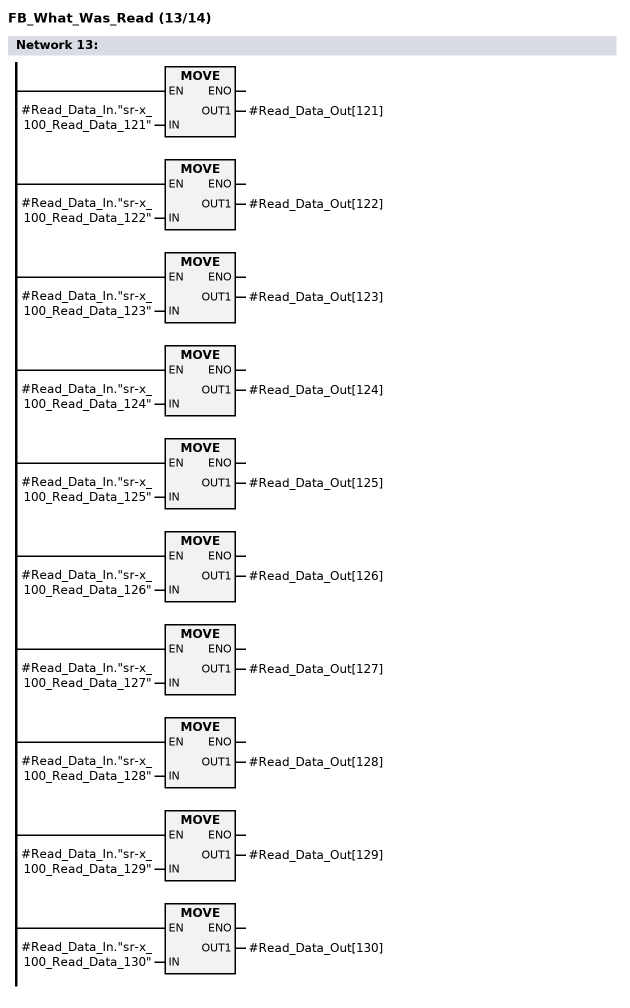
   RUNG wire#powerrail
      Move(in := #Read_Data_In."sr-x_100_Read_Data_121", out1 => #Read_Data_Out[121])
   END_RUNG
   RUNG wire#powerrail
      Move(in := #Read_Data_In."sr-x_100_Read_Data_122", out1 => #Read_Data_Out[122])
   END_RUNG
   RUNG wire#powerrail
      Move(in := #Read_Data_In."sr-x_100_Read_Data_123", out1 => #Read_Data_Out[123])
   END_RUNG
   RUNG wire#powerrail
      Move(in := #Read_Data_In."sr-x_100_Read_Data_124", out1 => #Read_Data_Out[124])
   END_RUNG
   RUNG wire#powerrail
      Move(in := #Read_Data_In."sr-x_100_Read_Data_125", out1 => #Read_Data_Out[125])
   END_RUNG
   RUNG wire#powerrail
      Move(in := #Read_Data_In."sr-x_100_Read_Data_126", out1 => #Read_Data_Out[126])
   END_RUNG
   RUNG wire#powerrail
      Move(in := #Read_Data_In."sr-x_100_Read_Data_127", out1 => #Read_Data_Out[127])
   END_RUNG
   RUNG wire#powerrail
      Move(in := #Read_Data_In."sr-x_100_Read_Data_128", out1 => #Read_Data_Out[128])
   END_RUNG
   RUNG wire#powerrail
      Move(in := #Read_Data_In."sr-x_100_Read_Data_129", out1 => #Read_Data_Out[129])
   END_RUNG
   RUNG wire#powerrail
      Move(in := #Read_Data_In."sr-x_100_Read_Data_130", out1 => #Read_Data_Out[130])
   END_RUNG
   // the same network as SCL:
   #Read_Data_Out[121] := #Read_Data_In."sr-x_100_Read_Data_121";
   #Read_Data_Out[122] := #Read_Data_In."sr-x_100_Read_Data_122";
   #Read_Data_Out[123] := #Read_Data_In."sr-x_100_Read_Data_123";
   #Read_Data_Out[124] := #Read_Data_In."sr-x_100_Read_Data_124";
   #Read_Data_Out[125] := #Read_Data_In."sr-x_100_Read_Data_125";
   #Read_Data_Out[126] := #Read_Data_In."sr-x_100_Read_Data_126";
   #Read_Data_Out[127] := #Read_Data_In."sr-x_100_Read_Data_127";
   #Read_Data_Out[128] := #Read_Data_In."sr-x_100_Read_Data_128";
   #Read_Data_Out[129] := #Read_Data_In."sr-x_100_Read_Data_129";
   #Read_Data_Out[130] := #Read_Data_In."sr-x_100_Read_Data_130";
END_REGION

REGION Network 14
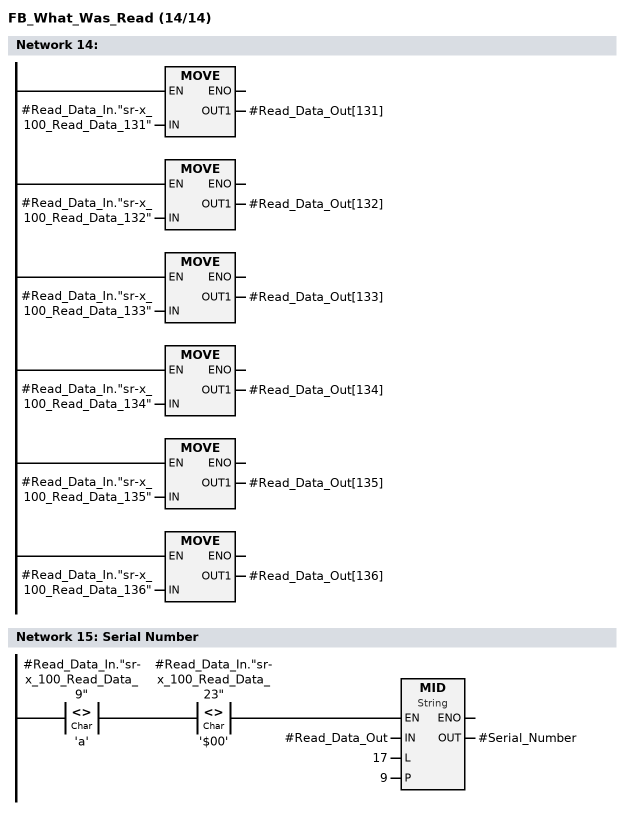
   RUNG wire#powerrail
      Move(in := #Read_Data_In."sr-x_100_Read_Data_131", out1 => #Read_Data_Out[131])
   END_RUNG
   RUNG wire#powerrail
      Move(in := #Read_Data_In."sr-x_100_Read_Data_132", out1 => #Read_Data_Out[132])
   END_RUNG
   RUNG wire#powerrail
      Move(in := #Read_Data_In."sr-x_100_Read_Data_133", out1 => #Read_Data_Out[133])
   END_RUNG
   RUNG wire#powerrail
      Move(in := #Read_Data_In."sr-x_100_Read_Data_134", out1 => #Read_Data_Out[134])
   END_RUNG
   RUNG wire#powerrail
      Move(in := #Read_Data_In."sr-x_100_Read_Data_135", out1 => #Read_Data_Out[135])
   END_RUNG
   RUNG wire#powerrail
      Move(in := #Read_Data_In."sr-x_100_Read_Data_136", out1 => #Read_Data_Out[136])
   END_RUNG
   // the same network as SCL:
   #Read_Data_Out[131] := #Read_Data_In."sr-x_100_Read_Data_131";
   #Read_Data_Out[132] := #Read_Data_In."sr-x_100_Read_Data_132";
   #Read_Data_Out[133] := #Read_Data_In."sr-x_100_Read_Data_133";
   #Read_Data_Out[134] := #Read_Data_In."sr-x_100_Read_Data_134";
   #Read_Data_Out[135] := #Read_Data_In."sr-x_100_Read_Data_135";
   #Read_Data_Out[136] := #Read_Data_In."sr-x_100_Read_Data_136";
END_REGION

REGION Network 15: Serial Number
   RUNG wire#powerrail
      { S7_Templates := "SrcType := Char" } NE_Contact(in1 := #Read_Data_In."sr-x_100_Read_Data_9", in2 := 'a')
      { S7_Templates := "SrcType := Char" } NE_Contact(in1 := #Read_Data_In."sr-x_100_Read_Data_23", in2 := '$00')
      { S7_Templates := "value_type := String" } MID(IN := #Read_Data_Out, L := 17, P := 9, OUT => #Serial_Number)
   END_RUNG
   // the same network as SCL:
   IF (#Read_Data_In."sr-x_100_Read_Data_9" <> 'a') AND (#Read_Data_In."sr-x_100_Read_Data_23" <> '$00') THEN
       MID(IN := #Read_Data_Out, L := 17, P := 9, OUT => #Serial_Number);
   END_IF;
END_REGION
END_FUNCTION_BLOCK

FUNCTION_BLOCK "FB_Marrige"   // FB8, LAD
{ S7_Optimized_Access := 'TRUE' }
// stored: MemoryReserve 100, SetENOAutomatically false
   VAR_INPUT
      In_Functional_Test_Odd : "IO_Device_Functinal_Test_Odd";
      In_Functional_Test_Even : "IO_Device_Functinal_Test_Even";
      Water_Fountain : String;
      Serial_Number : String[17];
      Read_Electrial_Voltage : UInt;
   END_VAR
   VAR_OUTPUT
      Functional_Tests_Panels : Array[0..31] of "Functional_Test";
      Got_Married : Bool;
   END_VAR
   VAR
      Aux_Trigger_0 : Bool;
      Aux_Trigger_1 : Bool;
      Aux_Trigger_2 : Bool;
      Aux_Trigger_3 : Bool;
      Aux_Trigger_4 : Bool;
      Aux_Trigger_5 : Bool;
      Aux_Trigger_6 : Bool;
      Aux_Trigger_7 : Bool;
      Aux_Trigger_8 : Bool;
      Aux_Trigger_9 : Bool;
      Aux_Trigger_10 : Bool;
      Aux_Trigger_11 : Bool;
      Aux_Trigger_12 : Bool;
      Aux_Trigger_13 : Bool;
      Aux_Trigger_14 : Bool;
      Aux_Trigger_15 : Bool;
      Aux_Trigger_16 : Bool;
      Aux_Trigger_17 : Bool;
      Aux_Trigger_18 : Bool;
      Aux_Trigger_19 : Bool;
      Aux_Trigger_20 : Bool;
      Aux_Trigger_21 : Bool;
      Aux_Trigger_22 : Bool;
      Aux_Trigger_23 : Bool;
      Aux_Trigger_24 : Bool;
      Aux_Trigger_25 : Bool;
      Aux_Trigger_26 : Bool;
      Aux_Trigger_27 : Bool;
      Aux_Trigger_28 : Bool;
      Aux_Trigger_29 : Bool;
      Aux_Trigger_30 : Bool;
      Aux_Trigger_31 : Bool;
   END_VAR
   VAR_TEMP   // added for the SCL form of the ladder/FBD networks
      _w1 : Bool;
   END_VAR
BEGIN

REGION Network 1: Panel 1
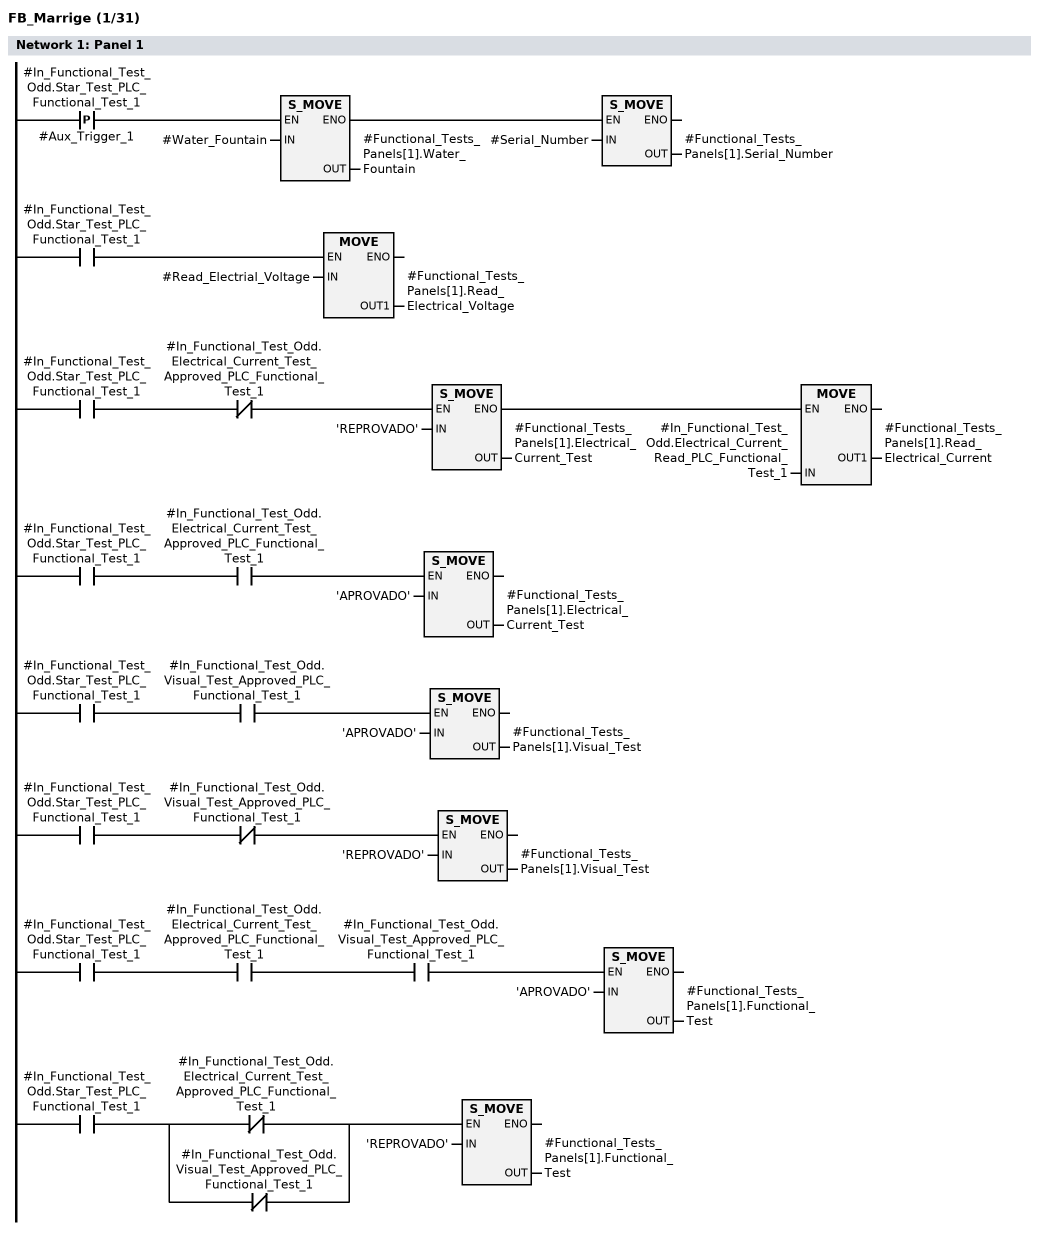
   RUNG wire#powerrail
      P_Contact(operand := #In_Functional_Test_Odd.Star_Test_PLC_Functional_Test_1, bit := #Aux_Trigger_1)
      S_Move(in := #Water_Fountain, out => #Functional_Tests_Panels[1].Water_Fountain)
      S_Move(in := #Serial_Number, out => #Functional_Tests_Panels[1].Serial_Number)
   END_RUNG
   RUNG wire#powerrail
      Contact( #In_Functional_Test_Odd.Star_Test_PLC_Functional_Test_1 )
      Move(in := #Read_Electrial_Voltage, out1 => #Functional_Tests_Panels[1].Read_Electrical_Voltage)
   END_RUNG
   RUNG wire#powerrail
      Contact( #In_Functional_Test_Odd.Star_Test_PLC_Functional_Test_1 )
      I_Contact( #In_Functional_Test_Odd.Electrical_Current_Test_Approved_PLC_Functional_Test_1 )
      S_Move(in := 'REPROVADO', out => #Functional_Tests_Panels[1].Electrical_Current_Test)
      Move(in := #In_Functional_Test_Odd.Electrical_Current_Read_PLC_Functional_Test_1, out1 => #Functional_Tests_Panels[1].Read_Electrical_Current)
   END_RUNG
   RUNG wire#powerrail
      Contact( #In_Functional_Test_Odd.Star_Test_PLC_Functional_Test_1 )
      Contact( #In_Functional_Test_Odd.Electrical_Current_Test_Approved_PLC_Functional_Test_1 )
      S_Move(in := 'APROVADO', out => #Functional_Tests_Panels[1].Electrical_Current_Test)
   END_RUNG
   RUNG wire#powerrail
      Contact( #In_Functional_Test_Odd.Star_Test_PLC_Functional_Test_1 )
      Contact( #In_Functional_Test_Odd.Visual_Test_Approved_PLC_Functional_Test_1 )
      S_Move(in := 'APROVADO', out => #Functional_Tests_Panels[1].Visual_Test)
   END_RUNG
   RUNG wire#powerrail
      Contact( #In_Functional_Test_Odd.Star_Test_PLC_Functional_Test_1 )
      I_Contact( #In_Functional_Test_Odd.Visual_Test_Approved_PLC_Functional_Test_1 )
      S_Move(in := 'REPROVADO', out => #Functional_Tests_Panels[1].Visual_Test)
   END_RUNG
   RUNG wire#powerrail
      Contact( #In_Functional_Test_Odd.Star_Test_PLC_Functional_Test_1 )
      Contact( #In_Functional_Test_Odd.Electrical_Current_Test_Approved_PLC_Functional_Test_1 )
      Contact( #In_Functional_Test_Odd.Visual_Test_Approved_PLC_Functional_Test_1 )
      S_Move(in := 'APROVADO', out => #Functional_Tests_Panels[1].Functional_Test)
   END_RUNG
   RUNG wire#powerrail
      Contact( #In_Functional_Test_Odd.Star_Test_PLC_Functional_Test_1 )
      wire#w1
      I_Contact( #In_Functional_Test_Odd.Electrical_Current_Test_Approved_PLC_Functional_Test_1 )
      wire#w2
      S_Move(in := 'REPROVADO', out => #Functional_Tests_Panels[1].Functional_Test)
   END_RUNG
   RUNG wire#w1
      I_Contact( #In_Functional_Test_Odd.Visual_Test_Approved_PLC_Functional_Test_1 )
   END_RUNG wire#w2
   // the same network as SCL:
   #_w1 := #In_Functional_Test_Odd.Star_Test_PLC_Functional_Test_1 AND NOT #Aux_Trigger_1;   // rising edge of #In_Functional_Test_Odd.Star_Test_PLC_Functional_Test_1
   #Aux_Trigger_1 := #In_Functional_Test_Odd.Star_Test_PLC_Functional_Test_1;
   IF #_w1 THEN
       #Functional_Tests_Panels[1].Water_Fountain := #Water_Fountain;
       #Functional_Tests_Panels[1].Serial_Number := #Serial_Number;
   END_IF;
   IF #In_Functional_Test_Odd.Star_Test_PLC_Functional_Test_1 THEN
       #Functional_Tests_Panels[1].Read_Electrical_Voltage := #Read_Electrial_Voltage;
   END_IF;
   IF #In_Functional_Test_Odd.Star_Test_PLC_Functional_Test_1 AND NOT #In_Functional_Test_Odd.Electrical_Current_Test_Approved_PLC_Functional_Test_1 THEN
       #Functional_Tests_Panels[1].Electrical_Current_Test := 'REPROVADO';
       #Functional_Tests_Panels[1].Read_Electrical_Current := #In_Functional_Test_Odd.Electrical_Current_Read_PLC_Functional_Test_1;
   END_IF;
   IF #In_Functional_Test_Odd.Star_Test_PLC_Functional_Test_1 AND #In_Functional_Test_Odd.Electrical_Current_Test_Approved_PLC_Functional_Test_1 THEN
       #Functional_Tests_Panels[1].Electrical_Current_Test := 'APROVADO';
   END_IF;
   IF #In_Functional_Test_Odd.Star_Test_PLC_Functional_Test_1 AND #In_Functional_Test_Odd.Visual_Test_Approved_PLC_Functional_Test_1 THEN
       #Functional_Tests_Panels[1].Visual_Test := 'APROVADO';
   END_IF;
   IF #In_Functional_Test_Odd.Star_Test_PLC_Functional_Test_1 AND NOT #In_Functional_Test_Odd.Visual_Test_Approved_PLC_Functional_Test_1 THEN
       #Functional_Tests_Panels[1].Visual_Test := 'REPROVADO';
   END_IF;
   IF #In_Functional_Test_Odd.Star_Test_PLC_Functional_Test_1 AND #In_Functional_Test_Odd.Electrical_Current_Test_Approved_PLC_Functional_Test_1 AND #In_Functional_Test_Odd.Visual_Test_Approved_PLC_Functional_Test_1 THEN
       #Functional_Tests_Panels[1].Functional_Test := 'APROVADO';
   END_IF;
   IF #In_Functional_Test_Odd.Star_Test_PLC_Functional_Test_1 AND (NOT #In_Functional_Test_Odd.Electrical_Current_Test_Approved_PLC_Functional_Test_1 OR NOT #In_Functional_Test_Odd.Visual_Test_Approved_PLC_Functional_Test_1) THEN
       #Functional_Tests_Panels[1].Functional_Test := 'REPROVADO';
   END_IF;
END_REGION

REGION Network 2: Panel 2
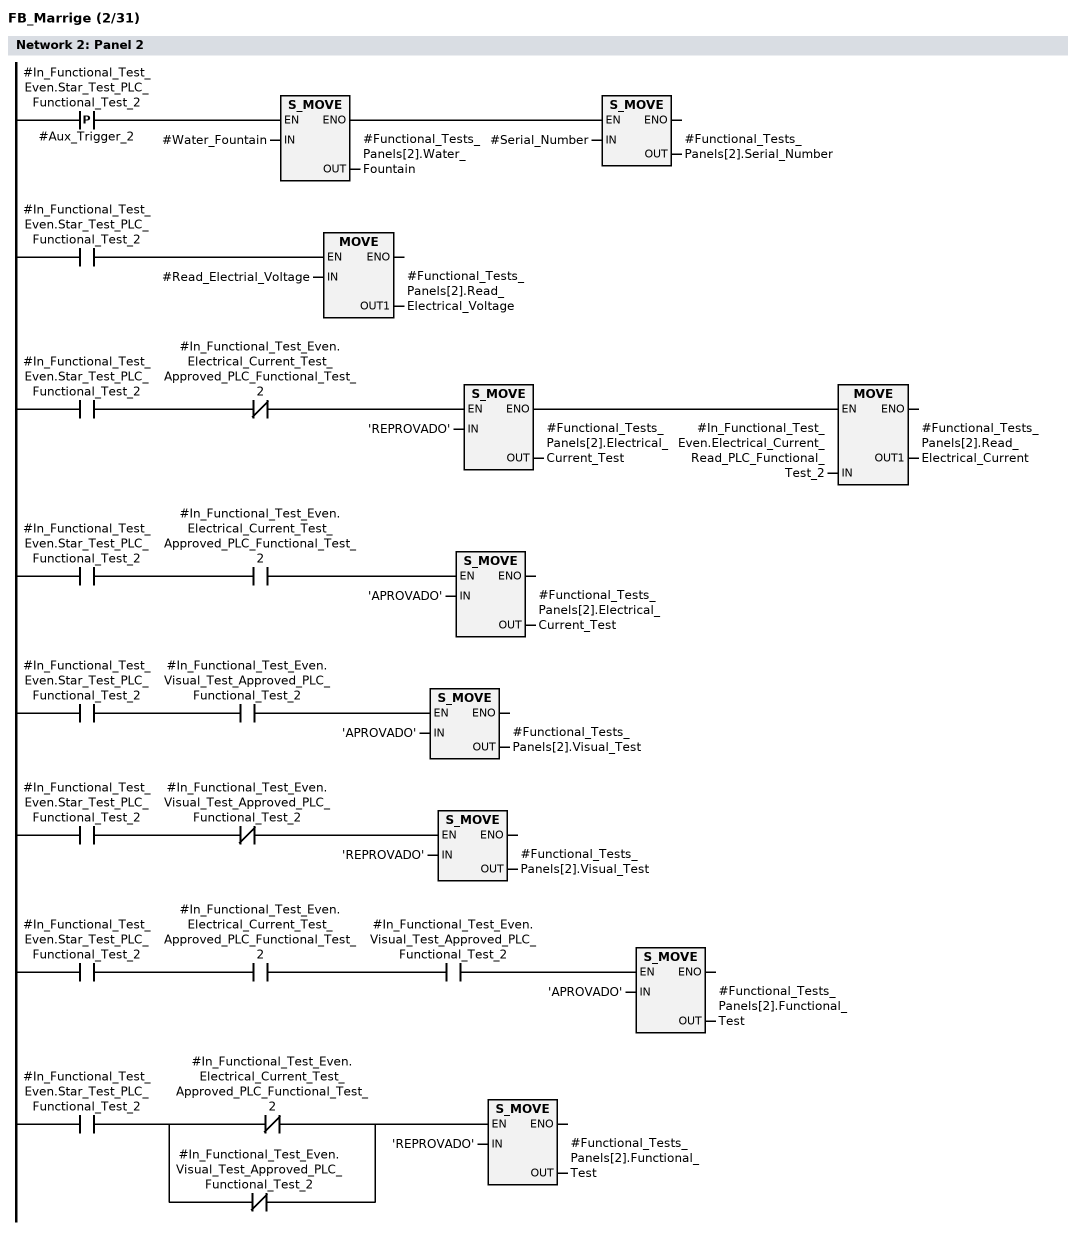
   RUNG wire#powerrail
      P_Contact(operand := #In_Functional_Test_Even.Star_Test_PLC_Functional_Test_2, bit := #Aux_Trigger_2)
      S_Move(in := #Water_Fountain, out => #Functional_Tests_Panels[2].Water_Fountain)
      S_Move(in := #Serial_Number, out => #Functional_Tests_Panels[2].Serial_Number)
   END_RUNG
   RUNG wire#powerrail
      Contact( #In_Functional_Test_Even.Star_Test_PLC_Functional_Test_2 )
      Move(in := #Read_Electrial_Voltage, out1 => #Functional_Tests_Panels[2].Read_Electrical_Voltage)
   END_RUNG
   RUNG wire#powerrail
      Contact( #In_Functional_Test_Even.Star_Test_PLC_Functional_Test_2 )
      I_Contact( #In_Functional_Test_Even.Electrical_Current_Test_Approved_PLC_Functional_Test_2 )
      S_Move(in := 'REPROVADO', out => #Functional_Tests_Panels[2].Electrical_Current_Test)
      Move(in := #In_Functional_Test_Even.Electrical_Current_Read_PLC_Functional_Test_2, out1 => #Functional_Tests_Panels[2].Read_Electrical_Current)
   END_RUNG
   RUNG wire#powerrail
      Contact( #In_Functional_Test_Even.Star_Test_PLC_Functional_Test_2 )
      Contact( #In_Functional_Test_Even.Electrical_Current_Test_Approved_PLC_Functional_Test_2 )
      S_Move(in := 'APROVADO', out => #Functional_Tests_Panels[2].Electrical_Current_Test)
   END_RUNG
   RUNG wire#powerrail
      Contact( #In_Functional_Test_Even.Star_Test_PLC_Functional_Test_2 )
      Contact( #In_Functional_Test_Even.Visual_Test_Approved_PLC_Functional_Test_2 )
      S_Move(in := 'APROVADO', out => #Functional_Tests_Panels[2].Visual_Test)
   END_RUNG
   RUNG wire#powerrail
      Contact( #In_Functional_Test_Even.Star_Test_PLC_Functional_Test_2 )
      I_Contact( #In_Functional_Test_Even.Visual_Test_Approved_PLC_Functional_Test_2 )
      S_Move(in := 'REPROVADO', out => #Functional_Tests_Panels[2].Visual_Test)
   END_RUNG
   RUNG wire#powerrail
      Contact( #In_Functional_Test_Even.Star_Test_PLC_Functional_Test_2 )
      Contact( #In_Functional_Test_Even.Electrical_Current_Test_Approved_PLC_Functional_Test_2 )
      Contact( #In_Functional_Test_Even.Visual_Test_Approved_PLC_Functional_Test_2 )
      S_Move(in := 'APROVADO', out => #Functional_Tests_Panels[2].Functional_Test)
   END_RUNG
   RUNG wire#powerrail
      Contact( #In_Functional_Test_Even.Star_Test_PLC_Functional_Test_2 )
      wire#w1
      I_Contact( #In_Functional_Test_Even.Electrical_Current_Test_Approved_PLC_Functional_Test_2 )
      wire#w2
      S_Move(in := 'REPROVADO', out => #Functional_Tests_Panels[2].Functional_Test)
   END_RUNG
   RUNG wire#w1
      I_Contact( #In_Functional_Test_Even.Visual_Test_Approved_PLC_Functional_Test_2 )
   END_RUNG wire#w2
   // the same network as SCL:
   #_w1 := #In_Functional_Test_Even.Star_Test_PLC_Functional_Test_2 AND NOT #Aux_Trigger_2;   // rising edge of #In_Functional_Test_Even.Star_Test_PLC_Functional_Test_2
   #Aux_Trigger_2 := #In_Functional_Test_Even.Star_Test_PLC_Functional_Test_2;
   IF #_w1 THEN
       #Functional_Tests_Panels[2].Water_Fountain := #Water_Fountain;
       #Functional_Tests_Panels[2].Serial_Number := #Serial_Number;
   END_IF;
   IF #In_Functional_Test_Even.Star_Test_PLC_Functional_Test_2 THEN
       #Functional_Tests_Panels[2].Read_Electrical_Voltage := #Read_Electrial_Voltage;
   END_IF;
   IF #In_Functional_Test_Even.Star_Test_PLC_Functional_Test_2 AND NOT #In_Functional_Test_Even.Electrical_Current_Test_Approved_PLC_Functional_Test_2 THEN
       #Functional_Tests_Panels[2].Electrical_Current_Test := 'REPROVADO';
       #Functional_Tests_Panels[2].Read_Electrical_Current := #In_Functional_Test_Even.Electrical_Current_Read_PLC_Functional_Test_2;
   END_IF;
   IF #In_Functional_Test_Even.Star_Test_PLC_Functional_Test_2 AND #In_Functional_Test_Even.Electrical_Current_Test_Approved_PLC_Functional_Test_2 THEN
       #Functional_Tests_Panels[2].Electrical_Current_Test := 'APROVADO';
   END_IF;
   IF #In_Functional_Test_Even.Star_Test_PLC_Functional_Test_2 AND #In_Functional_Test_Even.Visual_Test_Approved_PLC_Functional_Test_2 THEN
       #Functional_Tests_Panels[2].Visual_Test := 'APROVADO';
   END_IF;
   IF #In_Functional_Test_Even.Star_Test_PLC_Functional_Test_2 AND NOT #In_Functional_Test_Even.Visual_Test_Approved_PLC_Functional_Test_2 THEN
       #Functional_Tests_Panels[2].Visual_Test := 'REPROVADO';
   END_IF;
   IF #In_Functional_Test_Even.Star_Test_PLC_Functional_Test_2 AND #In_Functional_Test_Even.Electrical_Current_Test_Approved_PLC_Functional_Test_2 AND #In_Functional_Test_Even.Visual_Test_Approved_PLC_Functional_Test_2 THEN
       #Functional_Tests_Panels[2].Functional_Test := 'APROVADO';
   END_IF;
   IF #In_Functional_Test_Even.Star_Test_PLC_Functional_Test_2 AND (NOT #In_Functional_Test_Even.Electrical_Current_Test_Approved_PLC_Functional_Test_2 OR NOT #In_Functional_Test_Even.Visual_Test_Approved_PLC_Functional_Test_2) THEN
       #Functional_Tests_Panels[2].Functional_Test := 'REPROVADO';
   END_IF;
END_REGION

REGION Network 3: Panel 3
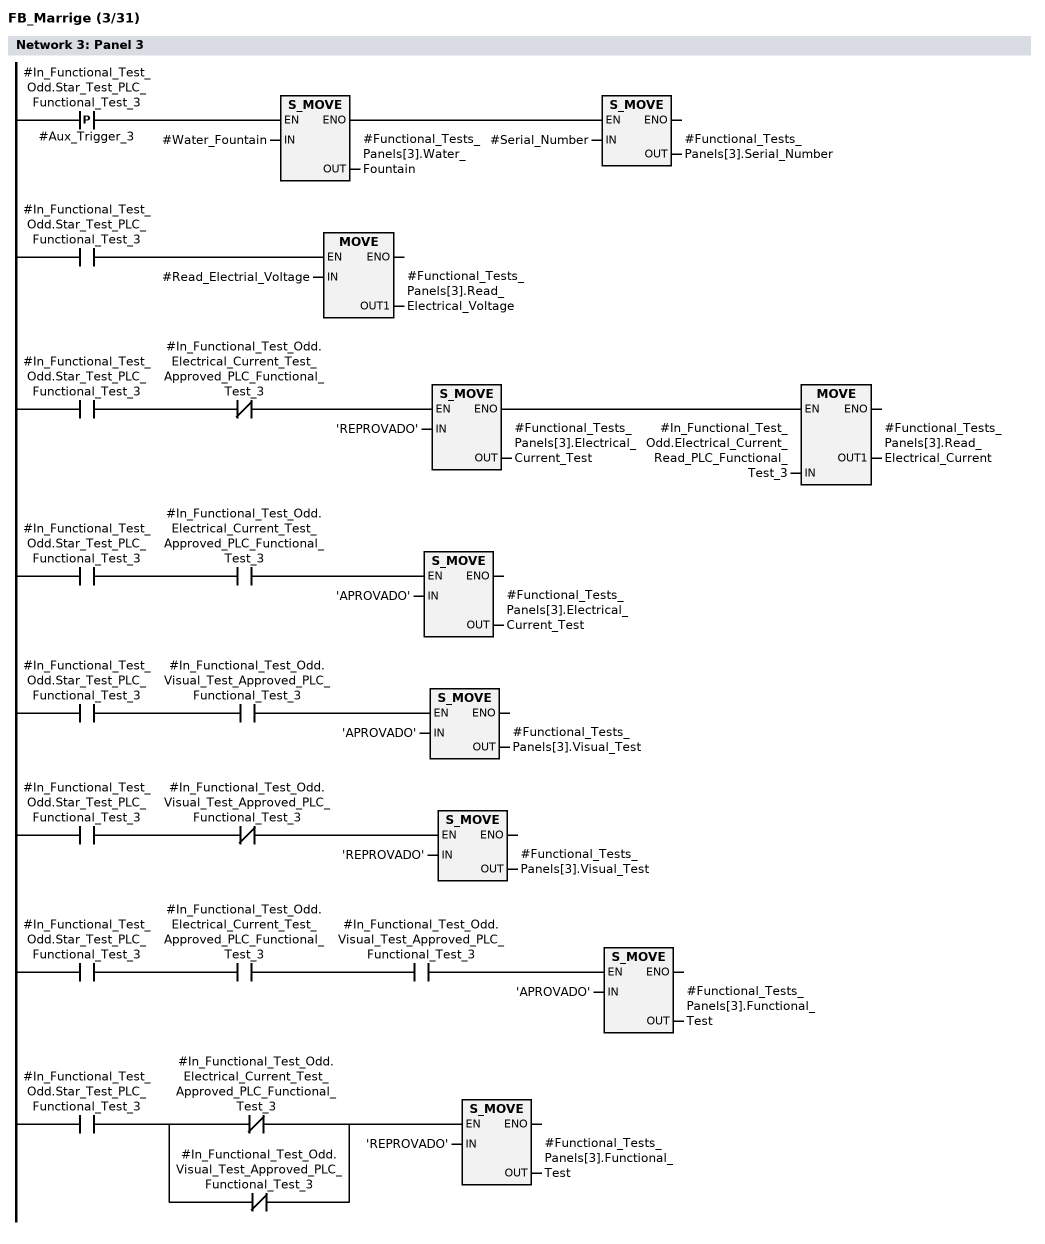
   RUNG wire#powerrail
      P_Contact(operand := #In_Functional_Test_Odd.Star_Test_PLC_Functional_Test_3, bit := #Aux_Trigger_3)
      S_Move(in := #Water_Fountain, out => #Functional_Tests_Panels[3].Water_Fountain)
      S_Move(in := #Serial_Number, out => #Functional_Tests_Panels[3].Serial_Number)
   END_RUNG
   RUNG wire#powerrail
      Contact( #In_Functional_Test_Odd.Star_Test_PLC_Functional_Test_3 )
      Move(in := #Read_Electrial_Voltage, out1 => #Functional_Tests_Panels[3].Read_Electrical_Voltage)
   END_RUNG
   RUNG wire#powerrail
      Contact( #In_Functional_Test_Odd.Star_Test_PLC_Functional_Test_3 )
      I_Contact( #In_Functional_Test_Odd.Electrical_Current_Test_Approved_PLC_Functional_Test_3 )
      S_Move(in := 'REPROVADO', out => #Functional_Tests_Panels[3].Electrical_Current_Test)
      Move(in := #In_Functional_Test_Odd.Electrical_Current_Read_PLC_Functional_Test_3, out1 => #Functional_Tests_Panels[3].Read_Electrical_Current)
   END_RUNG
   RUNG wire#powerrail
      Contact( #In_Functional_Test_Odd.Star_Test_PLC_Functional_Test_3 )
      Contact( #In_Functional_Test_Odd.Electrical_Current_Test_Approved_PLC_Functional_Test_3 )
      S_Move(in := 'APROVADO', out => #Functional_Tests_Panels[3].Electrical_Current_Test)
   END_RUNG
   RUNG wire#powerrail
      Contact( #In_Functional_Test_Odd.Star_Test_PLC_Functional_Test_3 )
      Contact( #In_Functional_Test_Odd.Visual_Test_Approved_PLC_Functional_Test_3 )
      S_Move(in := 'APROVADO', out => #Functional_Tests_Panels[3].Visual_Test)
   END_RUNG
   RUNG wire#powerrail
      Contact( #In_Functional_Test_Odd.Star_Test_PLC_Functional_Test_3 )
      I_Contact( #In_Functional_Test_Odd.Visual_Test_Approved_PLC_Functional_Test_3 )
      S_Move(in := 'REPROVADO', out => #Functional_Tests_Panels[3].Visual_Test)
   END_RUNG
   RUNG wire#powerrail
      Contact( #In_Functional_Test_Odd.Star_Test_PLC_Functional_Test_3 )
      Contact( #In_Functional_Test_Odd.Electrical_Current_Test_Approved_PLC_Functional_Test_3 )
      Contact( #In_Functional_Test_Odd.Visual_Test_Approved_PLC_Functional_Test_3 )
      S_Move(in := 'APROVADO', out => #Functional_Tests_Panels[3].Functional_Test)
   END_RUNG
   RUNG wire#powerrail
      Contact( #In_Functional_Test_Odd.Star_Test_PLC_Functional_Test_3 )
      wire#w1
      I_Contact( #In_Functional_Test_Odd.Electrical_Current_Test_Approved_PLC_Functional_Test_3 )
      wire#w2
      S_Move(in := 'REPROVADO', out => #Functional_Tests_Panels[3].Functional_Test)
   END_RUNG
   RUNG wire#w1
      I_Contact( #In_Functional_Test_Odd.Visual_Test_Approved_PLC_Functional_Test_3 )
   END_RUNG wire#w2
   // the same network as SCL:
   #_w1 := #In_Functional_Test_Odd.Star_Test_PLC_Functional_Test_3 AND NOT #Aux_Trigger_3;   // rising edge of #In_Functional_Test_Odd.Star_Test_PLC_Functional_Test_3
   #Aux_Trigger_3 := #In_Functional_Test_Odd.Star_Test_PLC_Functional_Test_3;
   IF #_w1 THEN
       #Functional_Tests_Panels[3].Water_Fountain := #Water_Fountain;
       #Functional_Tests_Panels[3].Serial_Number := #Serial_Number;
   END_IF;
   IF #In_Functional_Test_Odd.Star_Test_PLC_Functional_Test_3 THEN
       #Functional_Tests_Panels[3].Read_Electrical_Voltage := #Read_Electrial_Voltage;
   END_IF;
   IF #In_Functional_Test_Odd.Star_Test_PLC_Functional_Test_3 AND NOT #In_Functional_Test_Odd.Electrical_Current_Test_Approved_PLC_Functional_Test_3 THEN
       #Functional_Tests_Panels[3].Electrical_Current_Test := 'REPROVADO';
       #Functional_Tests_Panels[3].Read_Electrical_Current := #In_Functional_Test_Odd.Electrical_Current_Read_PLC_Functional_Test_3;
   END_IF;
   IF #In_Functional_Test_Odd.Star_Test_PLC_Functional_Test_3 AND #In_Functional_Test_Odd.Electrical_Current_Test_Approved_PLC_Functional_Test_3 THEN
       #Functional_Tests_Panels[3].Electrical_Current_Test := 'APROVADO';
   END_IF;
   IF #In_Functional_Test_Odd.Star_Test_PLC_Functional_Test_3 AND #In_Functional_Test_Odd.Visual_Test_Approved_PLC_Functional_Test_3 THEN
       #Functional_Tests_Panels[3].Visual_Test := 'APROVADO';
   END_IF;
   IF #In_Functional_Test_Odd.Star_Test_PLC_Functional_Test_3 AND NOT #In_Functional_Test_Odd.Visual_Test_Approved_PLC_Functional_Test_3 THEN
       #Functional_Tests_Panels[3].Visual_Test := 'REPROVADO';
   END_IF;
   IF #In_Functional_Test_Odd.Star_Test_PLC_Functional_Test_3 AND #In_Functional_Test_Odd.Electrical_Current_Test_Approved_PLC_Functional_Test_3 AND #In_Functional_Test_Odd.Visual_Test_Approved_PLC_Functional_Test_3 THEN
       #Functional_Tests_Panels[3].Functional_Test := 'APROVADO';
   END_IF;
   IF #In_Functional_Test_Odd.Star_Test_PLC_Functional_Test_3 AND (NOT #In_Functional_Test_Odd.Electrical_Current_Test_Approved_PLC_Functional_Test_3 OR NOT #In_Functional_Test_Odd.Visual_Test_Approved_PLC_Functional_Test_3) THEN
       #Functional_Tests_Panels[3].Functional_Test := 'REPROVADO';
   END_IF;
END_REGION

REGION Network 4: Panel 4
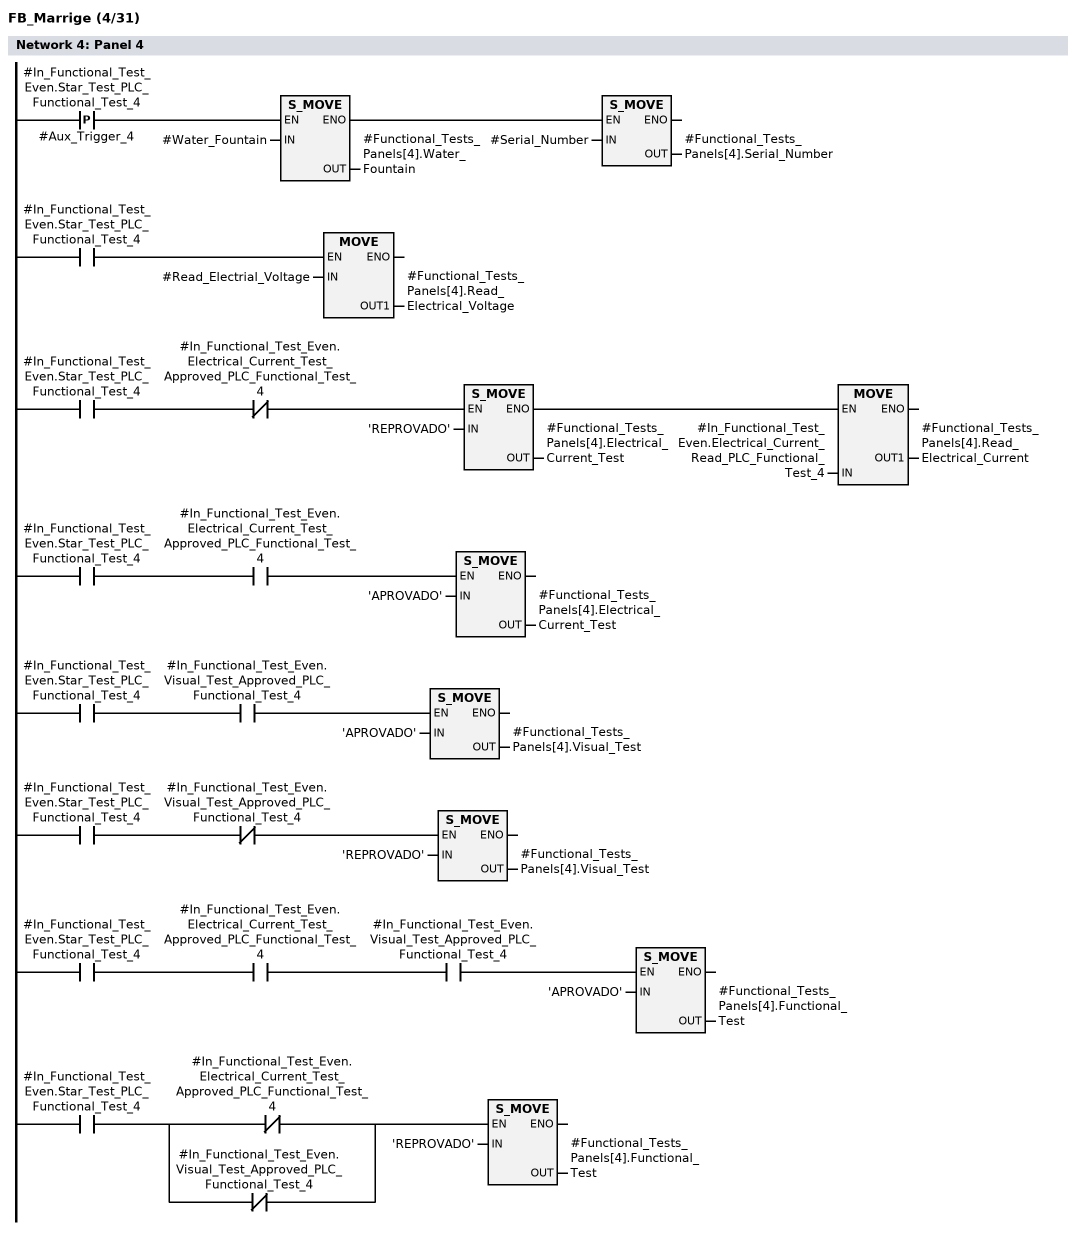
   RUNG wire#powerrail
      P_Contact(operand := #In_Functional_Test_Even.Star_Test_PLC_Functional_Test_4, bit := #Aux_Trigger_4)
      S_Move(in := #Water_Fountain, out => #Functional_Tests_Panels[4].Water_Fountain)
      S_Move(in := #Serial_Number, out => #Functional_Tests_Panels[4].Serial_Number)
   END_RUNG
   RUNG wire#powerrail
      Contact( #In_Functional_Test_Even.Star_Test_PLC_Functional_Test_4 )
      Move(in := #Read_Electrial_Voltage, out1 => #Functional_Tests_Panels[4].Read_Electrical_Voltage)
   END_RUNG
   RUNG wire#powerrail
      Contact( #In_Functional_Test_Even.Star_Test_PLC_Functional_Test_4 )
      I_Contact( #In_Functional_Test_Even.Electrical_Current_Test_Approved_PLC_Functional_Test_4 )
      S_Move(in := 'REPROVADO', out => #Functional_Tests_Panels[4].Electrical_Current_Test)
      Move(in := #In_Functional_Test_Even.Electrical_Current_Read_PLC_Functional_Test_4, out1 => #Functional_Tests_Panels[4].Read_Electrical_Current)
   END_RUNG
   RUNG wire#powerrail
      Contact( #In_Functional_Test_Even.Star_Test_PLC_Functional_Test_4 )
      Contact( #In_Functional_Test_Even.Electrical_Current_Test_Approved_PLC_Functional_Test_4 )
      S_Move(in := 'APROVADO', out => #Functional_Tests_Panels[4].Electrical_Current_Test)
   END_RUNG
   RUNG wire#powerrail
      Contact( #In_Functional_Test_Even.Star_Test_PLC_Functional_Test_4 )
      Contact( #In_Functional_Test_Even.Visual_Test_Approved_PLC_Functional_Test_4 )
      S_Move(in := 'APROVADO', out => #Functional_Tests_Panels[4].Visual_Test)
   END_RUNG
   RUNG wire#powerrail
      Contact( #In_Functional_Test_Even.Star_Test_PLC_Functional_Test_4 )
      I_Contact( #In_Functional_Test_Even.Visual_Test_Approved_PLC_Functional_Test_4 )
      S_Move(in := 'REPROVADO', out => #Functional_Tests_Panels[4].Visual_Test)
   END_RUNG
   RUNG wire#powerrail
      Contact( #In_Functional_Test_Even.Star_Test_PLC_Functional_Test_4 )
      Contact( #In_Functional_Test_Even.Electrical_Current_Test_Approved_PLC_Functional_Test_4 )
      Contact( #In_Functional_Test_Even.Visual_Test_Approved_PLC_Functional_Test_4 )
      S_Move(in := 'APROVADO', out => #Functional_Tests_Panels[4].Functional_Test)
   END_RUNG
   RUNG wire#powerrail
      Contact( #In_Functional_Test_Even.Star_Test_PLC_Functional_Test_4 )
      wire#w1
      I_Contact( #In_Functional_Test_Even.Electrical_Current_Test_Approved_PLC_Functional_Test_4 )
      wire#w2
      S_Move(in := 'REPROVADO', out => #Functional_Tests_Panels[4].Functional_Test)
   END_RUNG
   RUNG wire#w1
      I_Contact( #In_Functional_Test_Even.Visual_Test_Approved_PLC_Functional_Test_4 )
   END_RUNG wire#w2
   // the same network as SCL:
   #_w1 := #In_Functional_Test_Even.Star_Test_PLC_Functional_Test_4 AND NOT #Aux_Trigger_4;   // rising edge of #In_Functional_Test_Even.Star_Test_PLC_Functional_Test_4
   #Aux_Trigger_4 := #In_Functional_Test_Even.Star_Test_PLC_Functional_Test_4;
   IF #_w1 THEN
       #Functional_Tests_Panels[4].Water_Fountain := #Water_Fountain;
       #Functional_Tests_Panels[4].Serial_Number := #Serial_Number;
   END_IF;
   IF #In_Functional_Test_Even.Star_Test_PLC_Functional_Test_4 THEN
       #Functional_Tests_Panels[4].Read_Electrical_Voltage := #Read_Electrial_Voltage;
   END_IF;
   IF #In_Functional_Test_Even.Star_Test_PLC_Functional_Test_4 AND NOT #In_Functional_Test_Even.Electrical_Current_Test_Approved_PLC_Functional_Test_4 THEN
       #Functional_Tests_Panels[4].Electrical_Current_Test := 'REPROVADO';
       #Functional_Tests_Panels[4].Read_Electrical_Current := #In_Functional_Test_Even.Electrical_Current_Read_PLC_Functional_Test_4;
   END_IF;
   IF #In_Functional_Test_Even.Star_Test_PLC_Functional_Test_4 AND #In_Functional_Test_Even.Electrical_Current_Test_Approved_PLC_Functional_Test_4 THEN
       #Functional_Tests_Panels[4].Electrical_Current_Test := 'APROVADO';
   END_IF;
   IF #In_Functional_Test_Even.Star_Test_PLC_Functional_Test_4 AND #In_Functional_Test_Even.Visual_Test_Approved_PLC_Functional_Test_4 THEN
       #Functional_Tests_Panels[4].Visual_Test := 'APROVADO';
   END_IF;
   IF #In_Functional_Test_Even.Star_Test_PLC_Functional_Test_4 AND NOT #In_Functional_Test_Even.Visual_Test_Approved_PLC_Functional_Test_4 THEN
       #Functional_Tests_Panels[4].Visual_Test := 'REPROVADO';
   END_IF;
   IF #In_Functional_Test_Even.Star_Test_PLC_Functional_Test_4 AND #In_Functional_Test_Even.Electrical_Current_Test_Approved_PLC_Functional_Test_4 AND #In_Functional_Test_Even.Visual_Test_Approved_PLC_Functional_Test_4 THEN
       #Functional_Tests_Panels[4].Functional_Test := 'APROVADO';
   END_IF;
   IF #In_Functional_Test_Even.Star_Test_PLC_Functional_Test_4 AND (NOT #In_Functional_Test_Even.Electrical_Current_Test_Approved_PLC_Functional_Test_4 OR NOT #In_Functional_Test_Even.Visual_Test_Approved_PLC_Functional_Test_4) THEN
       #Functional_Tests_Panels[4].Functional_Test := 'REPROVADO';
   END_IF;
END_REGION

REGION Network 5: Panel 5
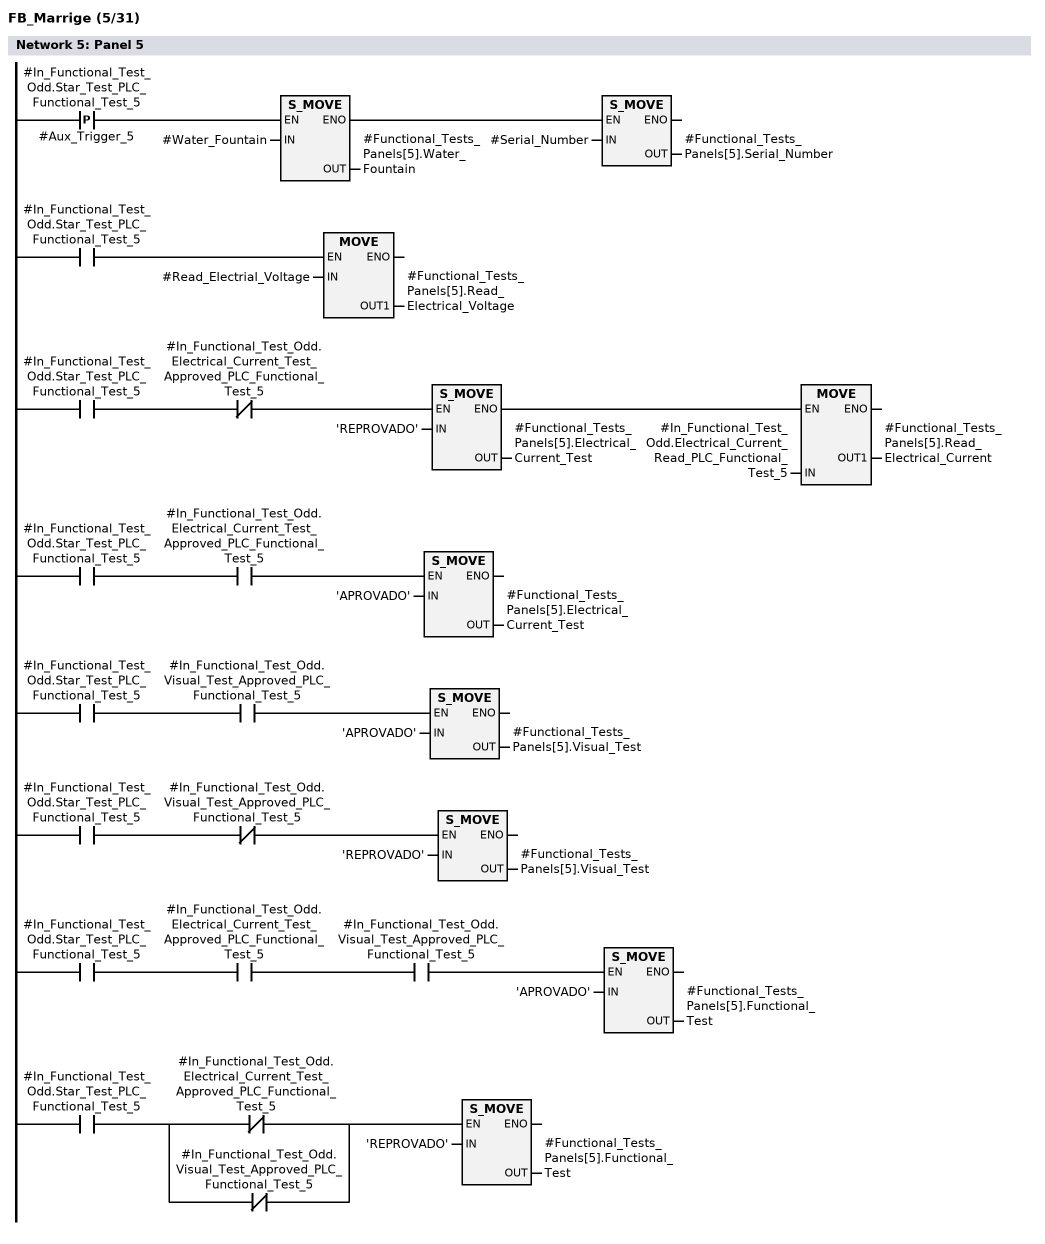
   RUNG wire#powerrail
      P_Contact(operand := #In_Functional_Test_Odd.Star_Test_PLC_Functional_Test_5, bit := #Aux_Trigger_5)
      S_Move(in := #Water_Fountain, out => #Functional_Tests_Panels[5].Water_Fountain)
      S_Move(in := #Serial_Number, out => #Functional_Tests_Panels[5].Serial_Number)
   END_RUNG
   RUNG wire#powerrail
      Contact( #In_Functional_Test_Odd.Star_Test_PLC_Functional_Test_5 )
      Move(in := #Read_Electrial_Voltage, out1 => #Functional_Tests_Panels[5].Read_Electrical_Voltage)
   END_RUNG
   RUNG wire#powerrail
      Contact( #In_Functional_Test_Odd.Star_Test_PLC_Functional_Test_5 )
      I_Contact( #In_Functional_Test_Odd.Electrical_Current_Test_Approved_PLC_Functional_Test_5 )
      S_Move(in := 'REPROVADO', out => #Functional_Tests_Panels[5].Electrical_Current_Test)
      Move(in := #In_Functional_Test_Odd.Electrical_Current_Read_PLC_Functional_Test_5, out1 => #Functional_Tests_Panels[5].Read_Electrical_Current)
   END_RUNG
   RUNG wire#powerrail
      Contact( #In_Functional_Test_Odd.Star_Test_PLC_Functional_Test_5 )
      Contact( #In_Functional_Test_Odd.Electrical_Current_Test_Approved_PLC_Functional_Test_5 )
      S_Move(in := 'APROVADO', out => #Functional_Tests_Panels[5].Electrical_Current_Test)
   END_RUNG
   RUNG wire#powerrail
      Contact( #In_Functional_Test_Odd.Star_Test_PLC_Functional_Test_5 )
      Contact( #In_Functional_Test_Odd.Visual_Test_Approved_PLC_Functional_Test_5 )
      S_Move(in := 'APROVADO', out => #Functional_Tests_Panels[5].Visual_Test)
   END_RUNG
   RUNG wire#powerrail
      Contact( #In_Functional_Test_Odd.Star_Test_PLC_Functional_Test_5 )
      I_Contact( #In_Functional_Test_Odd.Visual_Test_Approved_PLC_Functional_Test_5 )
      S_Move(in := 'REPROVADO', out => #Functional_Tests_Panels[5].Visual_Test)
   END_RUNG
   RUNG wire#powerrail
      Contact( #In_Functional_Test_Odd.Star_Test_PLC_Functional_Test_5 )
      Contact( #In_Functional_Test_Odd.Electrical_Current_Test_Approved_PLC_Functional_Test_5 )
      Contact( #In_Functional_Test_Odd.Visual_Test_Approved_PLC_Functional_Test_5 )
      S_Move(in := 'APROVADO', out => #Functional_Tests_Panels[5].Functional_Test)
   END_RUNG
   RUNG wire#powerrail
      Contact( #In_Functional_Test_Odd.Star_Test_PLC_Functional_Test_5 )
      wire#w1
      I_Contact( #In_Functional_Test_Odd.Electrical_Current_Test_Approved_PLC_Functional_Test_5 )
      wire#w2
      S_Move(in := 'REPROVADO', out => #Functional_Tests_Panels[5].Functional_Test)
   END_RUNG
   RUNG wire#w1
      I_Contact( #In_Functional_Test_Odd.Visual_Test_Approved_PLC_Functional_Test_5 )
   END_RUNG wire#w2
   // the same network as SCL:
   #_w1 := #In_Functional_Test_Odd.Star_Test_PLC_Functional_Test_5 AND NOT #Aux_Trigger_5;   // rising edge of #In_Functional_Test_Odd.Star_Test_PLC_Functional_Test_5
   #Aux_Trigger_5 := #In_Functional_Test_Odd.Star_Test_PLC_Functional_Test_5;
   IF #_w1 THEN
       #Functional_Tests_Panels[5].Water_Fountain := #Water_Fountain;
       #Functional_Tests_Panels[5].Serial_Number := #Serial_Number;
   END_IF;
   IF #In_Functional_Test_Odd.Star_Test_PLC_Functional_Test_5 THEN
       #Functional_Tests_Panels[5].Read_Electrical_Voltage := #Read_Electrial_Voltage;
   END_IF;
   IF #In_Functional_Test_Odd.Star_Test_PLC_Functional_Test_5 AND NOT #In_Functional_Test_Odd.Electrical_Current_Test_Approved_PLC_Functional_Test_5 THEN
       #Functional_Tests_Panels[5].Electrical_Current_Test := 'REPROVADO';
       #Functional_Tests_Panels[5].Read_Electrical_Current := #In_Functional_Test_Odd.Electrical_Current_Read_PLC_Functional_Test_5;
   END_IF;
   IF #In_Functional_Test_Odd.Star_Test_PLC_Functional_Test_5 AND #In_Functional_Test_Odd.Electrical_Current_Test_Approved_PLC_Functional_Test_5 THEN
       #Functional_Tests_Panels[5].Electrical_Current_Test := 'APROVADO';
   END_IF;
   IF #In_Functional_Test_Odd.Star_Test_PLC_Functional_Test_5 AND #In_Functional_Test_Odd.Visual_Test_Approved_PLC_Functional_Test_5 THEN
       #Functional_Tests_Panels[5].Visual_Test := 'APROVADO';
   END_IF;
   IF #In_Functional_Test_Odd.Star_Test_PLC_Functional_Test_5 AND NOT #In_Functional_Test_Odd.Visual_Test_Approved_PLC_Functional_Test_5 THEN
       #Functional_Tests_Panels[5].Visual_Test := 'REPROVADO';
   END_IF;
   IF #In_Functional_Test_Odd.Star_Test_PLC_Functional_Test_5 AND #In_Functional_Test_Odd.Electrical_Current_Test_Approved_PLC_Functional_Test_5 AND #In_Functional_Test_Odd.Visual_Test_Approved_PLC_Functional_Test_5 THEN
       #Functional_Tests_Panels[5].Functional_Test := 'APROVADO';
   END_IF;
   IF #In_Functional_Test_Odd.Star_Test_PLC_Functional_Test_5 AND (NOT #In_Functional_Test_Odd.Electrical_Current_Test_Approved_PLC_Functional_Test_5 OR NOT #In_Functional_Test_Odd.Visual_Test_Approved_PLC_Functional_Test_5) THEN
       #Functional_Tests_Panels[5].Functional_Test := 'REPROVADO';
   END_IF;
END_REGION

REGION Network 6: Panel 6
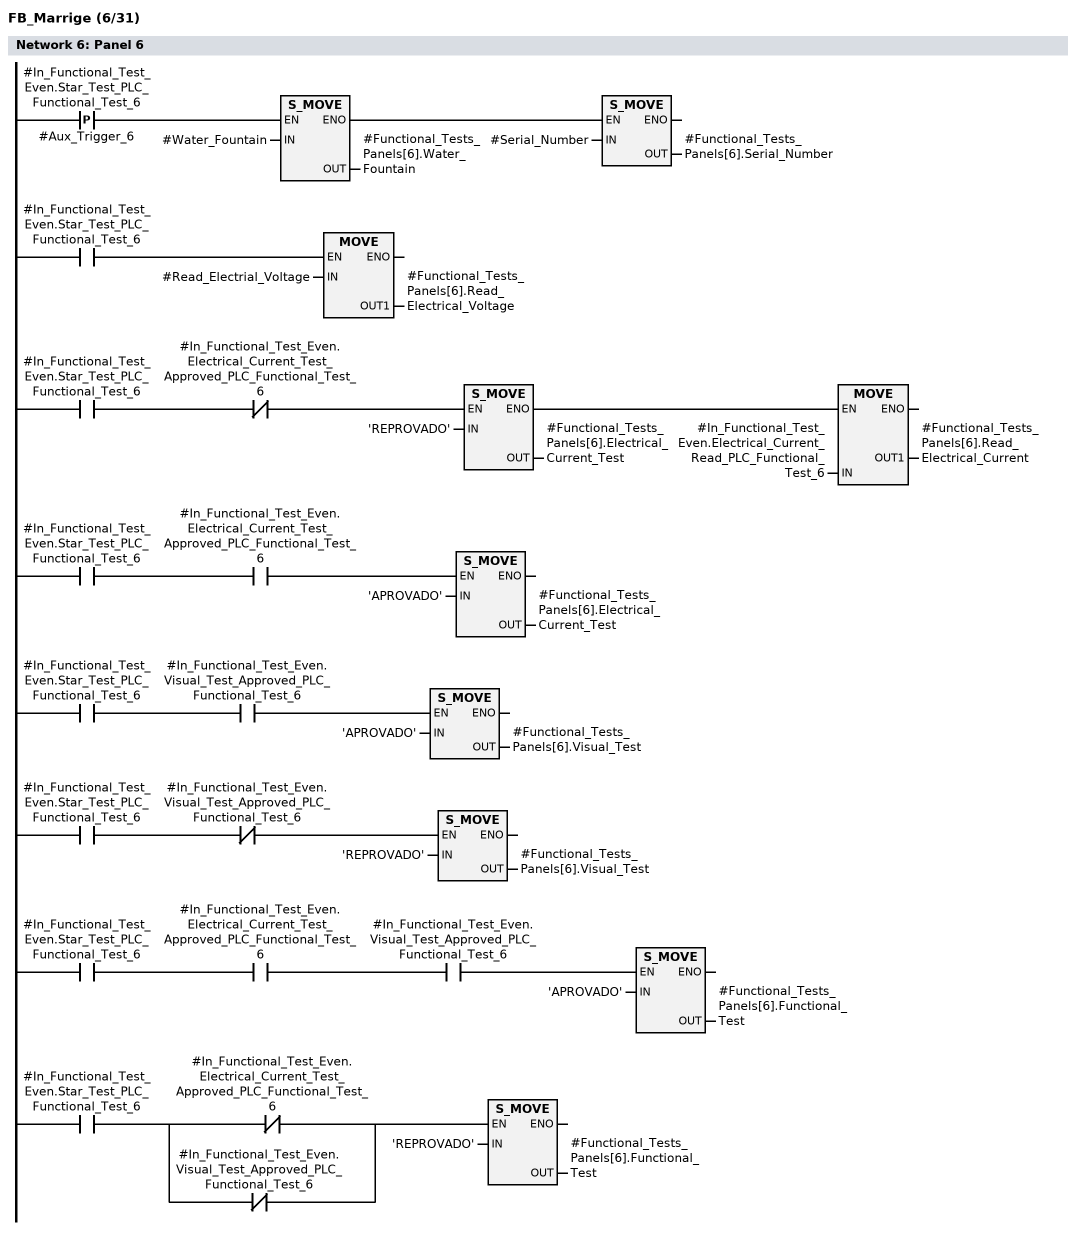
   RUNG wire#powerrail
      P_Contact(operand := #In_Functional_Test_Even.Star_Test_PLC_Functional_Test_6, bit := #Aux_Trigger_6)
      S_Move(in := #Water_Fountain, out => #Functional_Tests_Panels[6].Water_Fountain)
      S_Move(in := #Serial_Number, out => #Functional_Tests_Panels[6].Serial_Number)
   END_RUNG
   RUNG wire#powerrail
      Contact( #In_Functional_Test_Even.Star_Test_PLC_Functional_Test_6 )
      Move(in := #Read_Electrial_Voltage, out1 => #Functional_Tests_Panels[6].Read_Electrical_Voltage)
   END_RUNG
   RUNG wire#powerrail
      Contact( #In_Functional_Test_Even.Star_Test_PLC_Functional_Test_6 )
      I_Contact( #In_Functional_Test_Even.Electrical_Current_Test_Approved_PLC_Functional_Test_6 )
      S_Move(in := 'REPROVADO', out => #Functional_Tests_Panels[6].Electrical_Current_Test)
      Move(in := #In_Functional_Test_Even.Electrical_Current_Read_PLC_Functional_Test_6, out1 => #Functional_Tests_Panels[6].Read_Electrical_Current)
   END_RUNG
   RUNG wire#powerrail
      Contact( #In_Functional_Test_Even.Star_Test_PLC_Functional_Test_6 )
      Contact( #In_Functional_Test_Even.Electrical_Current_Test_Approved_PLC_Functional_Test_6 )
      S_Move(in := 'APROVADO', out => #Functional_Tests_Panels[6].Electrical_Current_Test)
   END_RUNG
   RUNG wire#powerrail
      Contact( #In_Functional_Test_Even.Star_Test_PLC_Functional_Test_6 )
      Contact( #In_Functional_Test_Even.Visual_Test_Approved_PLC_Functional_Test_6 )
      S_Move(in := 'APROVADO', out => #Functional_Tests_Panels[6].Visual_Test)
   END_RUNG
   RUNG wire#powerrail
      Contact( #In_Functional_Test_Even.Star_Test_PLC_Functional_Test_6 )
      I_Contact( #In_Functional_Test_Even.Visual_Test_Approved_PLC_Functional_Test_6 )
      S_Move(in := 'REPROVADO', out => #Functional_Tests_Panels[6].Visual_Test)
   END_RUNG
   RUNG wire#powerrail
      Contact( #In_Functional_Test_Even.Star_Test_PLC_Functional_Test_6 )
      Contact( #In_Functional_Test_Even.Electrical_Current_Test_Approved_PLC_Functional_Test_6 )
      Contact( #In_Functional_Test_Even.Visual_Test_Approved_PLC_Functional_Test_6 )
      S_Move(in := 'APROVADO', out => #Functional_Tests_Panels[6].Functional_Test)
   END_RUNG
   RUNG wire#powerrail
      Contact( #In_Functional_Test_Even.Star_Test_PLC_Functional_Test_6 )
      wire#w1
      I_Contact( #In_Functional_Test_Even.Electrical_Current_Test_Approved_PLC_Functional_Test_6 )
      wire#w2
      S_Move(in := 'REPROVADO', out => #Functional_Tests_Panels[6].Functional_Test)
   END_RUNG
   RUNG wire#w1
      I_Contact( #In_Functional_Test_Even.Visual_Test_Approved_PLC_Functional_Test_6 )
   END_RUNG wire#w2
   // the same network as SCL:
   #_w1 := #In_Functional_Test_Even.Star_Test_PLC_Functional_Test_6 AND NOT #Aux_Trigger_6;   // rising edge of #In_Functional_Test_Even.Star_Test_PLC_Functional_Test_6
   #Aux_Trigger_6 := #In_Functional_Test_Even.Star_Test_PLC_Functional_Test_6;
   IF #_w1 THEN
       #Functional_Tests_Panels[6].Water_Fountain := #Water_Fountain;
       #Functional_Tests_Panels[6].Serial_Number := #Serial_Number;
   END_IF;
   IF #In_Functional_Test_Even.Star_Test_PLC_Functional_Test_6 THEN
       #Functional_Tests_Panels[6].Read_Electrical_Voltage := #Read_Electrial_Voltage;
   END_IF;
   IF #In_Functional_Test_Even.Star_Test_PLC_Functional_Test_6 AND NOT #In_Functional_Test_Even.Electrical_Current_Test_Approved_PLC_Functional_Test_6 THEN
       #Functional_Tests_Panels[6].Electrical_Current_Test := 'REPROVADO';
       #Functional_Tests_Panels[6].Read_Electrical_Current := #In_Functional_Test_Even.Electrical_Current_Read_PLC_Functional_Test_6;
   END_IF;
   IF #In_Functional_Test_Even.Star_Test_PLC_Functional_Test_6 AND #In_Functional_Test_Even.Electrical_Current_Test_Approved_PLC_Functional_Test_6 THEN
       #Functional_Tests_Panels[6].Electrical_Current_Test := 'APROVADO';
   END_IF;
   IF #In_Functional_Test_Even.Star_Test_PLC_Functional_Test_6 AND #In_Functional_Test_Even.Visual_Test_Approved_PLC_Functional_Test_6 THEN
       #Functional_Tests_Panels[6].Visual_Test := 'APROVADO';
   END_IF;
   IF #In_Functional_Test_Even.Star_Test_PLC_Functional_Test_6 AND NOT #In_Functional_Test_Even.Visual_Test_Approved_PLC_Functional_Test_6 THEN
       #Functional_Tests_Panels[6].Visual_Test := 'REPROVADO';
   END_IF;
   IF #In_Functional_Test_Even.Star_Test_PLC_Functional_Test_6 AND #In_Functional_Test_Even.Electrical_Current_Test_Approved_PLC_Functional_Test_6 AND #In_Functional_Test_Even.Visual_Test_Approved_PLC_Functional_Test_6 THEN
       #Functional_Tests_Panels[6].Functional_Test := 'APROVADO';
   END_IF;
   IF #In_Functional_Test_Even.Star_Test_PLC_Functional_Test_6 AND (NOT #In_Functional_Test_Even.Electrical_Current_Test_Approved_PLC_Functional_Test_6 OR NOT #In_Functional_Test_Even.Visual_Test_Approved_PLC_Functional_Test_6) THEN
       #Functional_Tests_Panels[6].Functional_Test := 'REPROVADO';
   END_IF;
END_REGION

REGION Network 7: Panel 7
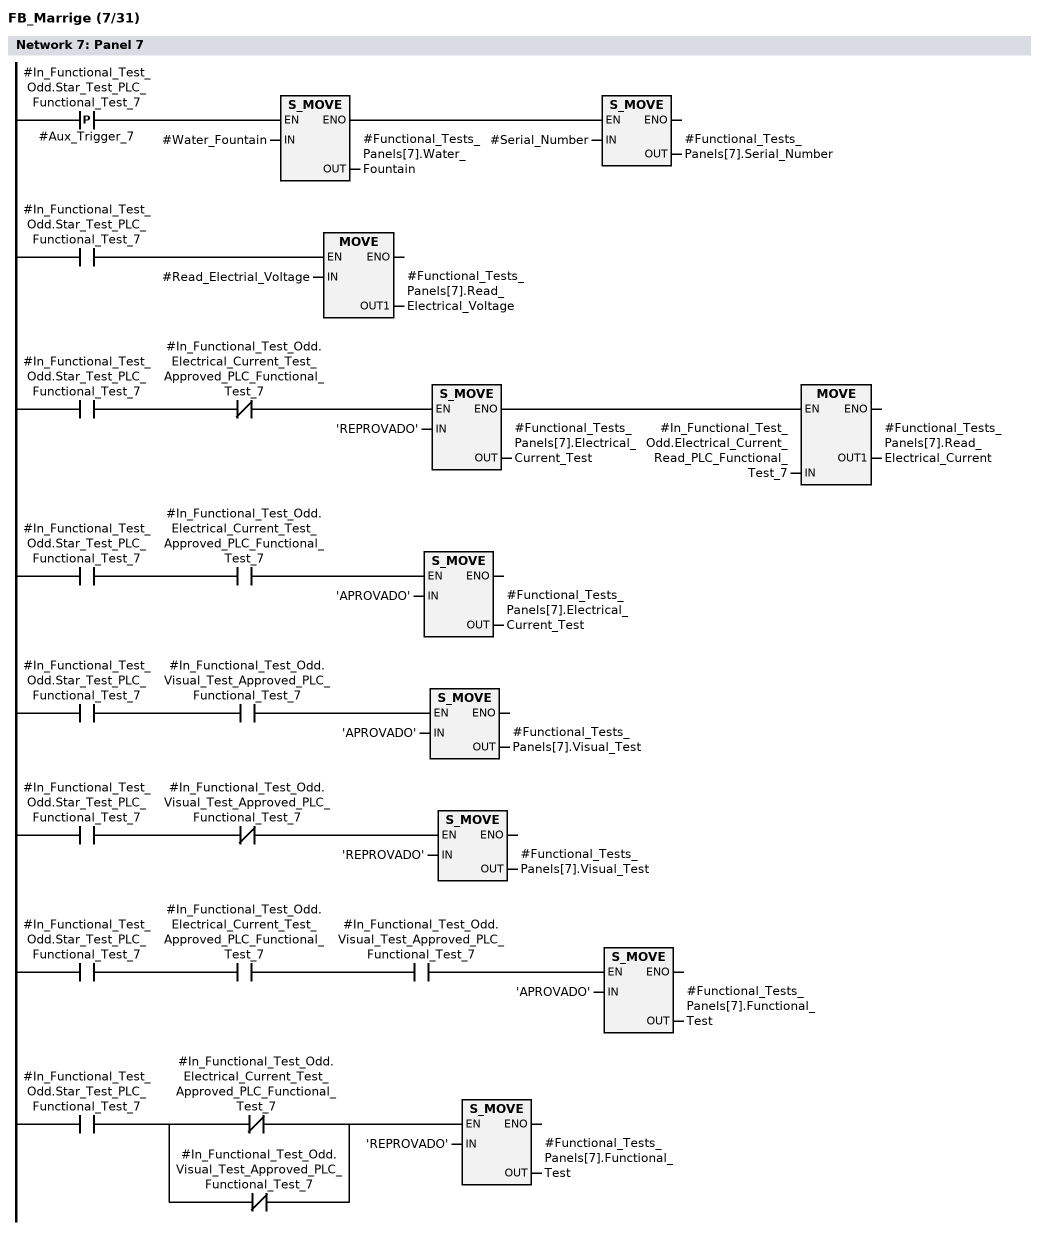
   RUNG wire#powerrail
      P_Contact(operand := #In_Functional_Test_Odd.Star_Test_PLC_Functional_Test_7, bit := #Aux_Trigger_7)
      S_Move(in := #Water_Fountain, out => #Functional_Tests_Panels[7].Water_Fountain)
      S_Move(in := #Serial_Number, out => #Functional_Tests_Panels[7].Serial_Number)
   END_RUNG
   RUNG wire#powerrail
      Contact( #In_Functional_Test_Odd.Star_Test_PLC_Functional_Test_7 )
      Move(in := #Read_Electrial_Voltage, out1 => #Functional_Tests_Panels[7].Read_Electrical_Voltage)
   END_RUNG
   RUNG wire#powerrail
      Contact( #In_Functional_Test_Odd.Star_Test_PLC_Functional_Test_7 )
      I_Contact( #In_Functional_Test_Odd.Electrical_Current_Test_Approved_PLC_Functional_Test_7 )
      S_Move(in := 'REPROVADO', out => #Functional_Tests_Panels[7].Electrical_Current_Test)
      Move(in := #In_Functional_Test_Odd.Electrical_Current_Read_PLC_Functional_Test_7, out1 => #Functional_Tests_Panels[7].Read_Electrical_Current)
   END_RUNG
   RUNG wire#powerrail
      Contact( #In_Functional_Test_Odd.Star_Test_PLC_Functional_Test_7 )
      Contact( #In_Functional_Test_Odd.Electrical_Current_Test_Approved_PLC_Functional_Test_7 )
      S_Move(in := 'APROVADO', out => #Functional_Tests_Panels[7].Electrical_Current_Test)
   END_RUNG
   RUNG wire#powerrail
      Contact( #In_Functional_Test_Odd.Star_Test_PLC_Functional_Test_7 )
      Contact( #In_Functional_Test_Odd.Visual_Test_Approved_PLC_Functional_Test_7 )
      S_Move(in := 'APROVADO', out => #Functional_Tests_Panels[7].Visual_Test)
   END_RUNG
   RUNG wire#powerrail
      Contact( #In_Functional_Test_Odd.Star_Test_PLC_Functional_Test_7 )
      I_Contact( #In_Functional_Test_Odd.Visual_Test_Approved_PLC_Functional_Test_7 )
      S_Move(in := 'REPROVADO', out => #Functional_Tests_Panels[7].Visual_Test)
   END_RUNG
   RUNG wire#powerrail
      Contact( #In_Functional_Test_Odd.Star_Test_PLC_Functional_Test_7 )
      Contact( #In_Functional_Test_Odd.Electrical_Current_Test_Approved_PLC_Functional_Test_7 )
      Contact( #In_Functional_Test_Odd.Visual_Test_Approved_PLC_Functional_Test_7 )
      S_Move(in := 'APROVADO', out => #Functional_Tests_Panels[7].Functional_Test)
   END_RUNG
   RUNG wire#powerrail
      Contact( #In_Functional_Test_Odd.Star_Test_PLC_Functional_Test_7 )
      wire#w1
      I_Contact( #In_Functional_Test_Odd.Electrical_Current_Test_Approved_PLC_Functional_Test_7 )
      wire#w2
      S_Move(in := 'REPROVADO', out => #Functional_Tests_Panels[7].Functional_Test)
   END_RUNG
   RUNG wire#w1
      I_Contact( #In_Functional_Test_Odd.Visual_Test_Approved_PLC_Functional_Test_7 )
   END_RUNG wire#w2
   // the same network as SCL:
   #_w1 := #In_Functional_Test_Odd.Star_Test_PLC_Functional_Test_7 AND NOT #Aux_Trigger_7;   // rising edge of #In_Functional_Test_Odd.Star_Test_PLC_Functional_Test_7
   #Aux_Trigger_7 := #In_Functional_Test_Odd.Star_Test_PLC_Functional_Test_7;
   IF #_w1 THEN
       #Functional_Tests_Panels[7].Water_Fountain := #Water_Fountain;
       #Functional_Tests_Panels[7].Serial_Number := #Serial_Number;
   END_IF;
   IF #In_Functional_Test_Odd.Star_Test_PLC_Functional_Test_7 THEN
       #Functional_Tests_Panels[7].Read_Electrical_Voltage := #Read_Electrial_Voltage;
   END_IF;
   IF #In_Functional_Test_Odd.Star_Test_PLC_Functional_Test_7 AND NOT #In_Functional_Test_Odd.Electrical_Current_Test_Approved_PLC_Functional_Test_7 THEN
       #Functional_Tests_Panels[7].Electrical_Current_Test := 'REPROVADO';
       #Functional_Tests_Panels[7].Read_Electrical_Current := #In_Functional_Test_Odd.Electrical_Current_Read_PLC_Functional_Test_7;
   END_IF;
   IF #In_Functional_Test_Odd.Star_Test_PLC_Functional_Test_7 AND #In_Functional_Test_Odd.Electrical_Current_Test_Approved_PLC_Functional_Test_7 THEN
       #Functional_Tests_Panels[7].Electrical_Current_Test := 'APROVADO';
   END_IF;
   IF #In_Functional_Test_Odd.Star_Test_PLC_Functional_Test_7 AND #In_Functional_Test_Odd.Visual_Test_Approved_PLC_Functional_Test_7 THEN
       #Functional_Tests_Panels[7].Visual_Test := 'APROVADO';
   END_IF;
   IF #In_Functional_Test_Odd.Star_Test_PLC_Functional_Test_7 AND NOT #In_Functional_Test_Odd.Visual_Test_Approved_PLC_Functional_Test_7 THEN
       #Functional_Tests_Panels[7].Visual_Test := 'REPROVADO';
   END_IF;
   IF #In_Functional_Test_Odd.Star_Test_PLC_Functional_Test_7 AND #In_Functional_Test_Odd.Electrical_Current_Test_Approved_PLC_Functional_Test_7 AND #In_Functional_Test_Odd.Visual_Test_Approved_PLC_Functional_Test_7 THEN
       #Functional_Tests_Panels[7].Functional_Test := 'APROVADO';
   END_IF;
   IF #In_Functional_Test_Odd.Star_Test_PLC_Functional_Test_7 AND (NOT #In_Functional_Test_Odd.Electrical_Current_Test_Approved_PLC_Functional_Test_7 OR NOT #In_Functional_Test_Odd.Visual_Test_Approved_PLC_Functional_Test_7) THEN
       #Functional_Tests_Panels[7].Functional_Test := 'REPROVADO';
   END_IF;
END_REGION

REGION Network 8: Panel 8
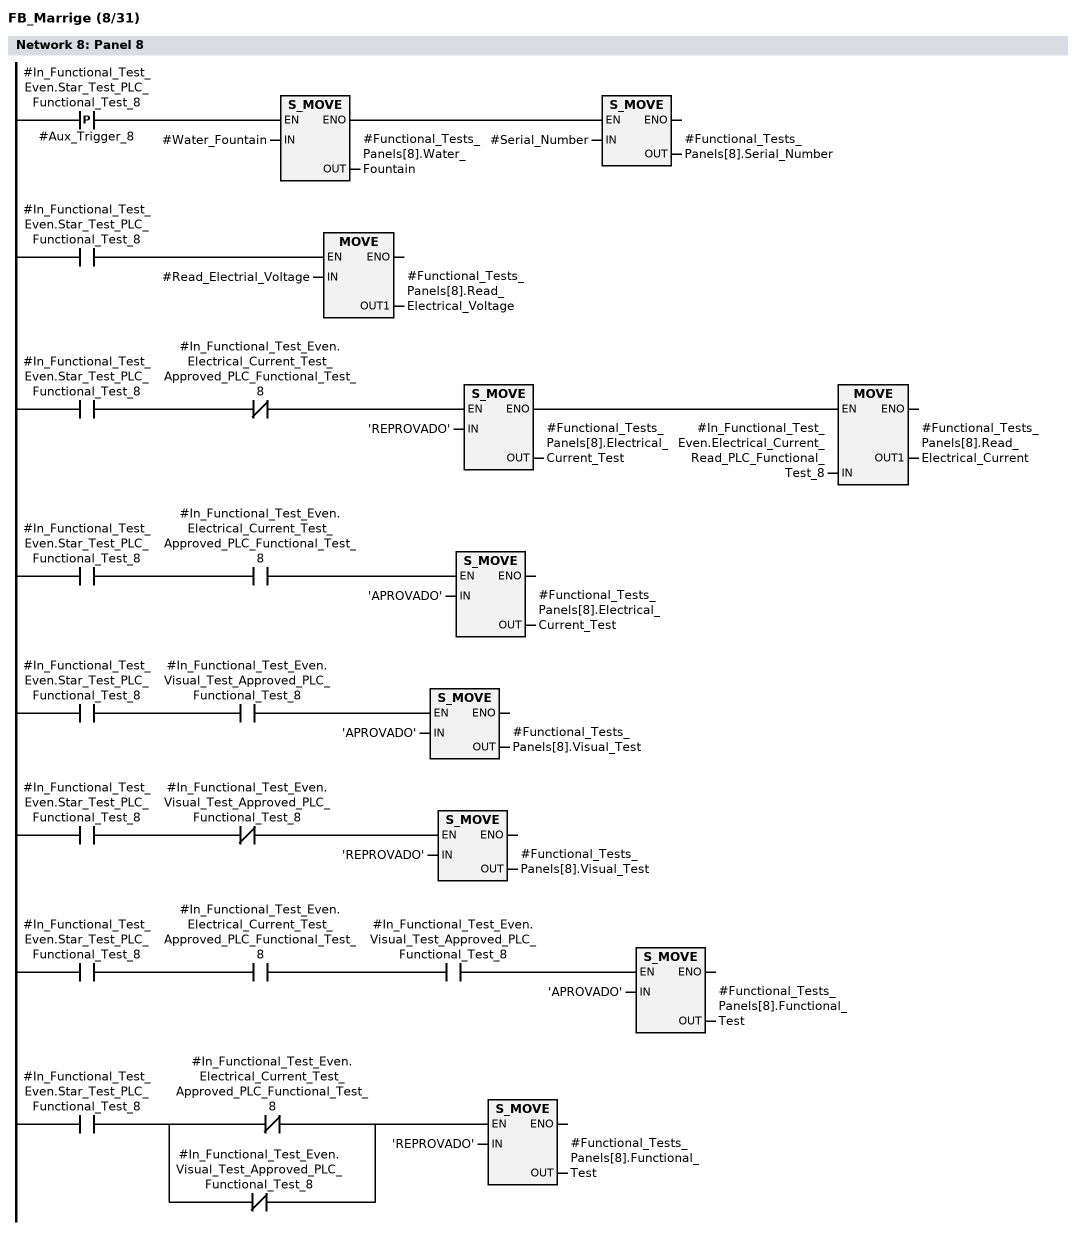
   RUNG wire#powerrail
      P_Contact(operand := #In_Functional_Test_Even.Star_Test_PLC_Functional_Test_8, bit := #Aux_Trigger_8)
      S_Move(in := #Water_Fountain, out => #Functional_Tests_Panels[8].Water_Fountain)
      S_Move(in := #Serial_Number, out => #Functional_Tests_Panels[8].Serial_Number)
   END_RUNG
   RUNG wire#powerrail
      Contact( #In_Functional_Test_Even.Star_Test_PLC_Functional_Test_8 )
      Move(in := #Read_Electrial_Voltage, out1 => #Functional_Tests_Panels[8].Read_Electrical_Voltage)
   END_RUNG
   RUNG wire#powerrail
      Contact( #In_Functional_Test_Even.Star_Test_PLC_Functional_Test_8 )
      I_Contact( #In_Functional_Test_Even.Electrical_Current_Test_Approved_PLC_Functional_Test_8 )
      S_Move(in := 'REPROVADO', out => #Functional_Tests_Panels[8].Electrical_Current_Test)
      Move(in := #In_Functional_Test_Even.Electrical_Current_Read_PLC_Functional_Test_8, out1 => #Functional_Tests_Panels[8].Read_Electrical_Current)
   END_RUNG
   RUNG wire#powerrail
      Contact( #In_Functional_Test_Even.Star_Test_PLC_Functional_Test_8 )
      Contact( #In_Functional_Test_Even.Electrical_Current_Test_Approved_PLC_Functional_Test_8 )
      S_Move(in := 'APROVADO', out => #Functional_Tests_Panels[8].Electrical_Current_Test)
   END_RUNG
   RUNG wire#powerrail
      Contact( #In_Functional_Test_Even.Star_Test_PLC_Functional_Test_8 )
      Contact( #In_Functional_Test_Even.Visual_Test_Approved_PLC_Functional_Test_8 )
      S_Move(in := 'APROVADO', out => #Functional_Tests_Panels[8].Visual_Test)
   END_RUNG
   RUNG wire#powerrail
      Contact( #In_Functional_Test_Even.Star_Test_PLC_Functional_Test_8 )
      I_Contact( #In_Functional_Test_Even.Visual_Test_Approved_PLC_Functional_Test_8 )
      S_Move(in := 'REPROVADO', out => #Functional_Tests_Panels[8].Visual_Test)
   END_RUNG
   RUNG wire#powerrail
      Contact( #In_Functional_Test_Even.Star_Test_PLC_Functional_Test_8 )
      Contact( #In_Functional_Test_Even.Electrical_Current_Test_Approved_PLC_Functional_Test_8 )
      Contact( #In_Functional_Test_Even.Visual_Test_Approved_PLC_Functional_Test_8 )
      S_Move(in := 'APROVADO', out => #Functional_Tests_Panels[8].Functional_Test)
   END_RUNG
   RUNG wire#powerrail
      Contact( #In_Functional_Test_Even.Star_Test_PLC_Functional_Test_8 )
      wire#w1
      I_Contact( #In_Functional_Test_Even.Electrical_Current_Test_Approved_PLC_Functional_Test_8 )
      wire#w2
      S_Move(in := 'REPROVADO', out => #Functional_Tests_Panels[8].Functional_Test)
   END_RUNG
   RUNG wire#w1
      I_Contact( #In_Functional_Test_Even.Visual_Test_Approved_PLC_Functional_Test_8 )
   END_RUNG wire#w2
   // the same network as SCL:
   #_w1 := #In_Functional_Test_Even.Star_Test_PLC_Functional_Test_8 AND NOT #Aux_Trigger_8;   // rising edge of #In_Functional_Test_Even.Star_Test_PLC_Functional_Test_8
   #Aux_Trigger_8 := #In_Functional_Test_Even.Star_Test_PLC_Functional_Test_8;
   IF #_w1 THEN
       #Functional_Tests_Panels[8].Water_Fountain := #Water_Fountain;
       #Functional_Tests_Panels[8].Serial_Number := #Serial_Number;
   END_IF;
   IF #In_Functional_Test_Even.Star_Test_PLC_Functional_Test_8 THEN
       #Functional_Tests_Panels[8].Read_Electrical_Voltage := #Read_Electrial_Voltage;
   END_IF;
   IF #In_Functional_Test_Even.Star_Test_PLC_Functional_Test_8 AND NOT #In_Functional_Test_Even.Electrical_Current_Test_Approved_PLC_Functional_Test_8 THEN
       #Functional_Tests_Panels[8].Electrical_Current_Test := 'REPROVADO';
       #Functional_Tests_Panels[8].Read_Electrical_Current := #In_Functional_Test_Even.Electrical_Current_Read_PLC_Functional_Test_8;
   END_IF;
   IF #In_Functional_Test_Even.Star_Test_PLC_Functional_Test_8 AND #In_Functional_Test_Even.Electrical_Current_Test_Approved_PLC_Functional_Test_8 THEN
       #Functional_Tests_Panels[8].Electrical_Current_Test := 'APROVADO';
   END_IF;
   IF #In_Functional_Test_Even.Star_Test_PLC_Functional_Test_8 AND #In_Functional_Test_Even.Visual_Test_Approved_PLC_Functional_Test_8 THEN
       #Functional_Tests_Panels[8].Visual_Test := 'APROVADO';
   END_IF;
   IF #In_Functional_Test_Even.Star_Test_PLC_Functional_Test_8 AND NOT #In_Functional_Test_Even.Visual_Test_Approved_PLC_Functional_Test_8 THEN
       #Functional_Tests_Panels[8].Visual_Test := 'REPROVADO';
   END_IF;
   IF #In_Functional_Test_Even.Star_Test_PLC_Functional_Test_8 AND #In_Functional_Test_Even.Electrical_Current_Test_Approved_PLC_Functional_Test_8 AND #In_Functional_Test_Even.Visual_Test_Approved_PLC_Functional_Test_8 THEN
       #Functional_Tests_Panels[8].Functional_Test := 'APROVADO';
   END_IF;
   IF #In_Functional_Test_Even.Star_Test_PLC_Functional_Test_8 AND (NOT #In_Functional_Test_Even.Electrical_Current_Test_Approved_PLC_Functional_Test_8 OR NOT #In_Functional_Test_Even.Visual_Test_Approved_PLC_Functional_Test_8) THEN
       #Functional_Tests_Panels[8].Functional_Test := 'REPROVADO';
   END_IF;
END_REGION

REGION Network 9: Panel 9
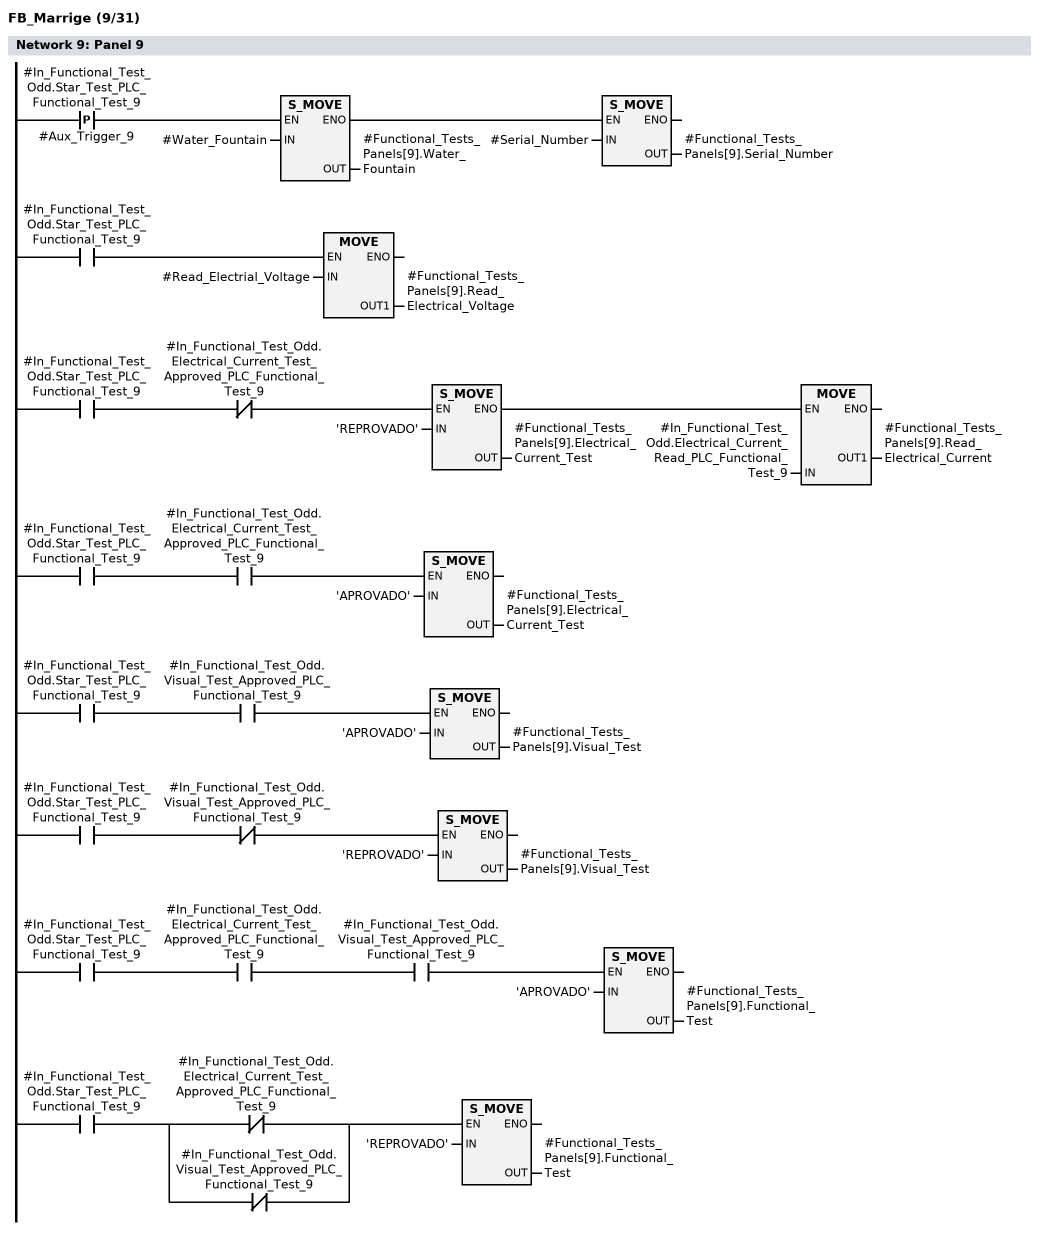
   RUNG wire#powerrail
      P_Contact(operand := #In_Functional_Test_Odd.Star_Test_PLC_Functional_Test_9, bit := #Aux_Trigger_9)
      S_Move(in := #Water_Fountain, out => #Functional_Tests_Panels[9].Water_Fountain)
      S_Move(in := #Serial_Number, out => #Functional_Tests_Panels[9].Serial_Number)
   END_RUNG
   RUNG wire#powerrail
      Contact( #In_Functional_Test_Odd.Star_Test_PLC_Functional_Test_9 )
      Move(in := #Read_Electrial_Voltage, out1 => #Functional_Tests_Panels[9].Read_Electrical_Voltage)
   END_RUNG
   RUNG wire#powerrail
      Contact( #In_Functional_Test_Odd.Star_Test_PLC_Functional_Test_9 )
      I_Contact( #In_Functional_Test_Odd.Electrical_Current_Test_Approved_PLC_Functional_Test_9 )
      S_Move(in := 'REPROVADO', out => #Functional_Tests_Panels[9].Electrical_Current_Test)
      Move(in := #In_Functional_Test_Odd.Electrical_Current_Read_PLC_Functional_Test_9, out1 => #Functional_Tests_Panels[9].Read_Electrical_Current)
   END_RUNG
   RUNG wire#powerrail
      Contact( #In_Functional_Test_Odd.Star_Test_PLC_Functional_Test_9 )
      Contact( #In_Functional_Test_Odd.Electrical_Current_Test_Approved_PLC_Functional_Test_9 )
      S_Move(in := 'APROVADO', out => #Functional_Tests_Panels[9].Electrical_Current_Test)
   END_RUNG
   RUNG wire#powerrail
      Contact( #In_Functional_Test_Odd.Star_Test_PLC_Functional_Test_9 )
      Contact( #In_Functional_Test_Odd.Visual_Test_Approved_PLC_Functional_Test_9 )
      S_Move(in := 'APROVADO', out => #Functional_Tests_Panels[9].Visual_Test)
   END_RUNG
   RUNG wire#powerrail
      Contact( #In_Functional_Test_Odd.Star_Test_PLC_Functional_Test_9 )
      I_Contact( #In_Functional_Test_Odd.Visual_Test_Approved_PLC_Functional_Test_9 )
      S_Move(in := 'REPROVADO', out => #Functional_Tests_Panels[9].Visual_Test)
   END_RUNG
   RUNG wire#powerrail
      Contact( #In_Functional_Test_Odd.Star_Test_PLC_Functional_Test_9 )
      Contact( #In_Functional_Test_Odd.Electrical_Current_Test_Approved_PLC_Functional_Test_9 )
      Contact( #In_Functional_Test_Odd.Visual_Test_Approved_PLC_Functional_Test_9 )
      S_Move(in := 'APROVADO', out => #Functional_Tests_Panels[9].Functional_Test)
   END_RUNG
   RUNG wire#powerrail
      Contact( #In_Functional_Test_Odd.Star_Test_PLC_Functional_Test_9 )
      wire#w1
      I_Contact( #In_Functional_Test_Odd.Electrical_Current_Test_Approved_PLC_Functional_Test_9 )
      wire#w2
      S_Move(in := 'REPROVADO', out => #Functional_Tests_Panels[9].Functional_Test)
   END_RUNG
   RUNG wire#w1
      I_Contact( #In_Functional_Test_Odd.Visual_Test_Approved_PLC_Functional_Test_9 )
   END_RUNG wire#w2
   // the same network as SCL:
   #_w1 := #In_Functional_Test_Odd.Star_Test_PLC_Functional_Test_9 AND NOT #Aux_Trigger_9;   // rising edge of #In_Functional_Test_Odd.Star_Test_PLC_Functional_Test_9
   #Aux_Trigger_9 := #In_Functional_Test_Odd.Star_Test_PLC_Functional_Test_9;
   IF #_w1 THEN
       #Functional_Tests_Panels[9].Water_Fountain := #Water_Fountain;
       #Functional_Tests_Panels[9].Serial_Number := #Serial_Number;
   END_IF;
   IF #In_Functional_Test_Odd.Star_Test_PLC_Functional_Test_9 THEN
       #Functional_Tests_Panels[9].Read_Electrical_Voltage := #Read_Electrial_Voltage;
   END_IF;
   IF #In_Functional_Test_Odd.Star_Test_PLC_Functional_Test_9 AND NOT #In_Functional_Test_Odd.Electrical_Current_Test_Approved_PLC_Functional_Test_9 THEN
       #Functional_Tests_Panels[9].Electrical_Current_Test := 'REPROVADO';
       #Functional_Tests_Panels[9].Read_Electrical_Current := #In_Functional_Test_Odd.Electrical_Current_Read_PLC_Functional_Test_9;
   END_IF;
   IF #In_Functional_Test_Odd.Star_Test_PLC_Functional_Test_9 AND #In_Functional_Test_Odd.Electrical_Current_Test_Approved_PLC_Functional_Test_9 THEN
       #Functional_Tests_Panels[9].Electrical_Current_Test := 'APROVADO';
   END_IF;
   IF #In_Functional_Test_Odd.Star_Test_PLC_Functional_Test_9 AND #In_Functional_Test_Odd.Visual_Test_Approved_PLC_Functional_Test_9 THEN
       #Functional_Tests_Panels[9].Visual_Test := 'APROVADO';
   END_IF;
   IF #In_Functional_Test_Odd.Star_Test_PLC_Functional_Test_9 AND NOT #In_Functional_Test_Odd.Visual_Test_Approved_PLC_Functional_Test_9 THEN
       #Functional_Tests_Panels[9].Visual_Test := 'REPROVADO';
   END_IF;
   IF #In_Functional_Test_Odd.Star_Test_PLC_Functional_Test_9 AND #In_Functional_Test_Odd.Electrical_Current_Test_Approved_PLC_Functional_Test_9 AND #In_Functional_Test_Odd.Visual_Test_Approved_PLC_Functional_Test_9 THEN
       #Functional_Tests_Panels[9].Functional_Test := 'APROVADO';
   END_IF;
   IF #In_Functional_Test_Odd.Star_Test_PLC_Functional_Test_9 AND (NOT #In_Functional_Test_Odd.Electrical_Current_Test_Approved_PLC_Functional_Test_9 OR NOT #In_Functional_Test_Odd.Visual_Test_Approved_PLC_Functional_Test_9) THEN
       #Functional_Tests_Panels[9].Functional_Test := 'REPROVADO';
   END_IF;
END_REGION

REGION Network 10: Panel 10
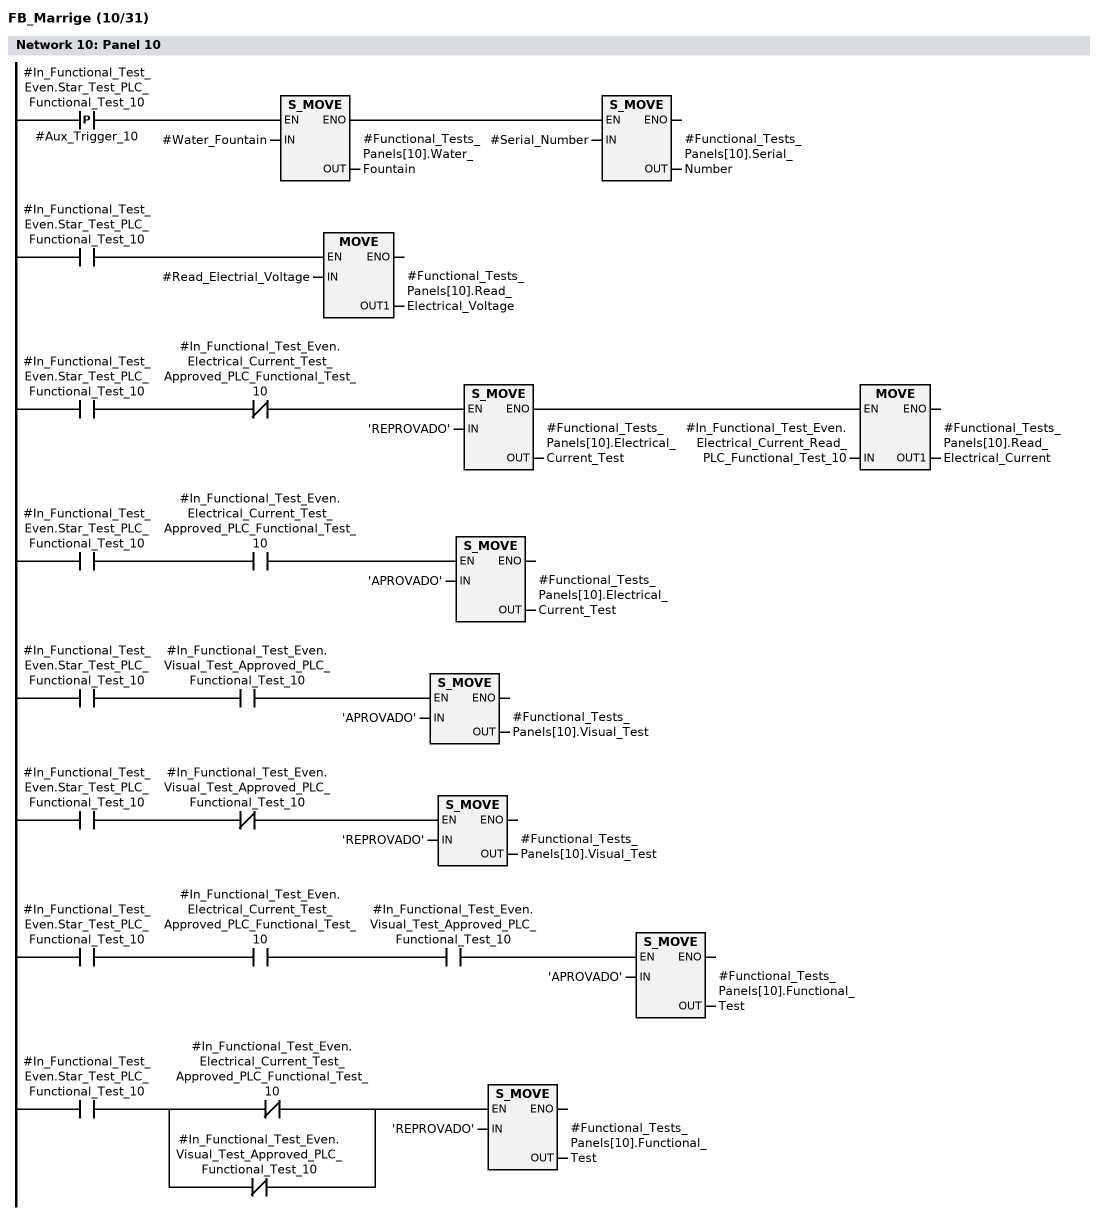
   RUNG wire#powerrail
      P_Contact(operand := #In_Functional_Test_Even.Star_Test_PLC_Functional_Test_10, bit := #Aux_Trigger_10)
      S_Move(in := #Water_Fountain, out => #Functional_Tests_Panels[10].Water_Fountain)
      S_Move(in := #Serial_Number, out => #Functional_Tests_Panels[10].Serial_Number)
   END_RUNG
   RUNG wire#powerrail
      Contact( #In_Functional_Test_Even.Star_Test_PLC_Functional_Test_10 )
      Move(in := #Read_Electrial_Voltage, out1 => #Functional_Tests_Panels[10].Read_Electrical_Voltage)
   END_RUNG
   RUNG wire#powerrail
      Contact( #In_Functional_Test_Even.Star_Test_PLC_Functional_Test_10 )
      I_Contact( #In_Functional_Test_Even.Electrical_Current_Test_Approved_PLC_Functional_Test_10 )
      S_Move(in := 'REPROVADO', out => #Functional_Tests_Panels[10].Electrical_Current_Test)
      Move(in := #In_Functional_Test_Even.Electrical_Current_Read_PLC_Functional_Test_10, out1 => #Functional_Tests_Panels[10].Read_Electrical_Current)
   END_RUNG
   RUNG wire#powerrail
      Contact( #In_Functional_Test_Even.Star_Test_PLC_Functional_Test_10 )
      Contact( #In_Functional_Test_Even.Electrical_Current_Test_Approved_PLC_Functional_Test_10 )
      S_Move(in := 'APROVADO', out => #Functional_Tests_Panels[10].Electrical_Current_Test)
   END_RUNG
   RUNG wire#powerrail
      Contact( #In_Functional_Test_Even.Star_Test_PLC_Functional_Test_10 )
      Contact( #In_Functional_Test_Even.Visual_Test_Approved_PLC_Functional_Test_10 )
      S_Move(in := 'APROVADO', out => #Functional_Tests_Panels[10].Visual_Test)
   END_RUNG
   RUNG wire#powerrail
      Contact( #In_Functional_Test_Even.Star_Test_PLC_Functional_Test_10 )
      I_Contact( #In_Functional_Test_Even.Visual_Test_Approved_PLC_Functional_Test_10 )
      S_Move(in := 'REPROVADO', out => #Functional_Tests_Panels[10].Visual_Test)
   END_RUNG
   RUNG wire#powerrail
      Contact( #In_Functional_Test_Even.Star_Test_PLC_Functional_Test_10 )
      Contact( #In_Functional_Test_Even.Electrical_Current_Test_Approved_PLC_Functional_Test_10 )
      Contact( #In_Functional_Test_Even.Visual_Test_Approved_PLC_Functional_Test_10 )
      S_Move(in := 'APROVADO', out => #Functional_Tests_Panels[10].Functional_Test)
   END_RUNG
   RUNG wire#powerrail
      Contact( #In_Functional_Test_Even.Star_Test_PLC_Functional_Test_10 )
      wire#w1
      I_Contact( #In_Functional_Test_Even.Electrical_Current_Test_Approved_PLC_Functional_Test_10 )
      wire#w2
      S_Move(in := 'REPROVADO', out => #Functional_Tests_Panels[10].Functional_Test)
   END_RUNG
   RUNG wire#w1
      I_Contact( #In_Functional_Test_Even.Visual_Test_Approved_PLC_Functional_Test_10 )
   END_RUNG wire#w2
   // the same network as SCL:
   #_w1 := #In_Functional_Test_Even.Star_Test_PLC_Functional_Test_10 AND NOT #Aux_Trigger_10;   // rising edge of #In_Functional_Test_Even.Star_Test_PLC_Functional_Test_10
   #Aux_Trigger_10 := #In_Functional_Test_Even.Star_Test_PLC_Functional_Test_10;
   IF #_w1 THEN
       #Functional_Tests_Panels[10].Water_Fountain := #Water_Fountain;
       #Functional_Tests_Panels[10].Serial_Number := #Serial_Number;
   END_IF;
   IF #In_Functional_Test_Even.Star_Test_PLC_Functional_Test_10 THEN
       #Functional_Tests_Panels[10].Read_Electrical_Voltage := #Read_Electrial_Voltage;
   END_IF;
   IF #In_Functional_Test_Even.Star_Test_PLC_Functional_Test_10 AND NOT #In_Functional_Test_Even.Electrical_Current_Test_Approved_PLC_Functional_Test_10 THEN
       #Functional_Tests_Panels[10].Electrical_Current_Test := 'REPROVADO';
       #Functional_Tests_Panels[10].Read_Electrical_Current := #In_Functional_Test_Even.Electrical_Current_Read_PLC_Functional_Test_10;
   END_IF;
   IF #In_Functional_Test_Even.Star_Test_PLC_Functional_Test_10 AND #In_Functional_Test_Even.Electrical_Current_Test_Approved_PLC_Functional_Test_10 THEN
       #Functional_Tests_Panels[10].Electrical_Current_Test := 'APROVADO';
   END_IF;
   IF #In_Functional_Test_Even.Star_Test_PLC_Functional_Test_10 AND #In_Functional_Test_Even.Visual_Test_Approved_PLC_Functional_Test_10 THEN
       #Functional_Tests_Panels[10].Visual_Test := 'APROVADO';
   END_IF;
   IF #In_Functional_Test_Even.Star_Test_PLC_Functional_Test_10 AND NOT #In_Functional_Test_Even.Visual_Test_Approved_PLC_Functional_Test_10 THEN
       #Functional_Tests_Panels[10].Visual_Test := 'REPROVADO';
   END_IF;
   IF #In_Functional_Test_Even.Star_Test_PLC_Functional_Test_10 AND #In_Functional_Test_Even.Electrical_Current_Test_Approved_PLC_Functional_Test_10 AND #In_Functional_Test_Even.Visual_Test_Approved_PLC_Functional_Test_10 THEN
       #Functional_Tests_Panels[10].Functional_Test := 'APROVADO';
   END_IF;
   IF #In_Functional_Test_Even.Star_Test_PLC_Functional_Test_10 AND (NOT #In_Functional_Test_Even.Electrical_Current_Test_Approved_PLC_Functional_Test_10 OR NOT #In_Functional_Test_Even.Visual_Test_Approved_PLC_Functional_Test_10) THEN
       #Functional_Tests_Panels[10].Functional_Test := 'REPROVADO';
   END_IF;
END_REGION

REGION Network 11: Panel 11
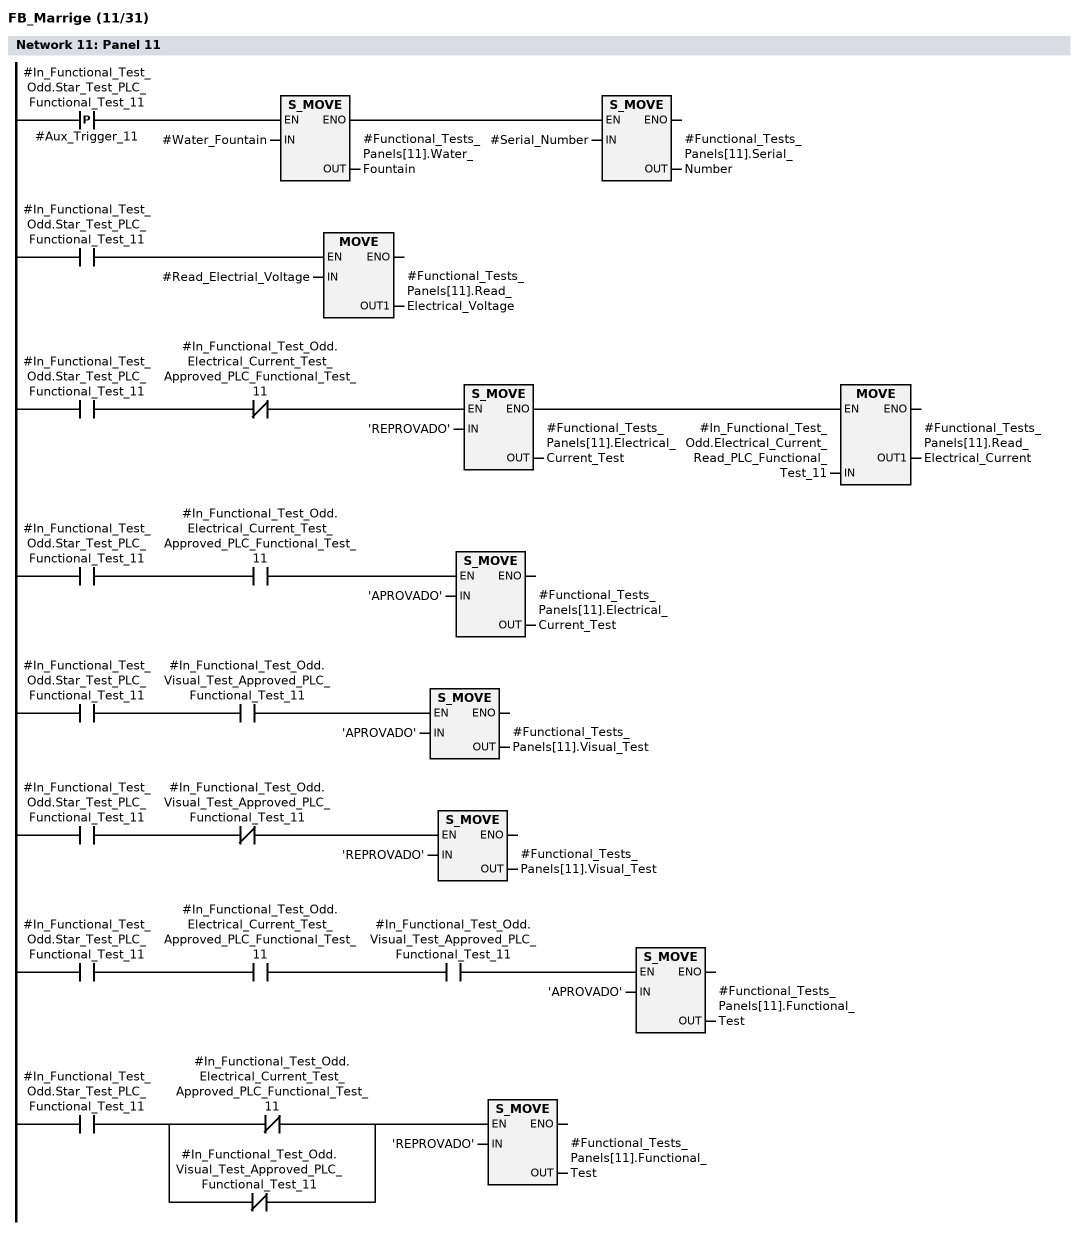
   RUNG wire#powerrail
      P_Contact(operand := #In_Functional_Test_Odd.Star_Test_PLC_Functional_Test_11, bit := #Aux_Trigger_11)
      S_Move(in := #Water_Fountain, out => #Functional_Tests_Panels[11].Water_Fountain)
      S_Move(in := #Serial_Number, out => #Functional_Tests_Panels[11].Serial_Number)
   END_RUNG
   RUNG wire#powerrail
      Contact( #In_Functional_Test_Odd.Star_Test_PLC_Functional_Test_11 )
      Move(in := #Read_Electrial_Voltage, out1 => #Functional_Tests_Panels[11].Read_Electrical_Voltage)
   END_RUNG
   RUNG wire#powerrail
      Contact( #In_Functional_Test_Odd.Star_Test_PLC_Functional_Test_11 )
      I_Contact( #In_Functional_Test_Odd.Electrical_Current_Test_Approved_PLC_Functional_Test_11 )
      S_Move(in := 'REPROVADO', out => #Functional_Tests_Panels[11].Electrical_Current_Test)
      Move(in := #In_Functional_Test_Odd.Electrical_Current_Read_PLC_Functional_Test_11, out1 => #Functional_Tests_Panels[11].Read_Electrical_Current)
   END_RUNG
   RUNG wire#powerrail
      Contact( #In_Functional_Test_Odd.Star_Test_PLC_Functional_Test_11 )
      Contact( #In_Functional_Test_Odd.Electrical_Current_Test_Approved_PLC_Functional_Test_11 )
      S_Move(in := 'APROVADO', out => #Functional_Tests_Panels[11].Electrical_Current_Test)
   END_RUNG
   RUNG wire#powerrail
      Contact( #In_Functional_Test_Odd.Star_Test_PLC_Functional_Test_11 )
      Contact( #In_Functional_Test_Odd.Visual_Test_Approved_PLC_Functional_Test_11 )
      S_Move(in := 'APROVADO', out => #Functional_Tests_Panels[11].Visual_Test)
   END_RUNG
   RUNG wire#powerrail
      Contact( #In_Functional_Test_Odd.Star_Test_PLC_Functional_Test_11 )
      I_Contact( #In_Functional_Test_Odd.Visual_Test_Approved_PLC_Functional_Test_11 )
      S_Move(in := 'REPROVADO', out => #Functional_Tests_Panels[11].Visual_Test)
   END_RUNG
   RUNG wire#powerrail
      Contact( #In_Functional_Test_Odd.Star_Test_PLC_Functional_Test_11 )
      Contact( #In_Functional_Test_Odd.Electrical_Current_Test_Approved_PLC_Functional_Test_11 )
      Contact( #In_Functional_Test_Odd.Visual_Test_Approved_PLC_Functional_Test_11 )
      S_Move(in := 'APROVADO', out => #Functional_Tests_Panels[11].Functional_Test)
   END_RUNG
   RUNG wire#powerrail
      Contact( #In_Functional_Test_Odd.Star_Test_PLC_Functional_Test_11 )
      wire#w1
      I_Contact( #In_Functional_Test_Odd.Electrical_Current_Test_Approved_PLC_Functional_Test_11 )
      wire#w2
      S_Move(in := 'REPROVADO', out => #Functional_Tests_Panels[11].Functional_Test)
   END_RUNG
   RUNG wire#w1
      I_Contact( #In_Functional_Test_Odd.Visual_Test_Approved_PLC_Functional_Test_11 )
   END_RUNG wire#w2
   // the same network as SCL:
   #_w1 := #In_Functional_Test_Odd.Star_Test_PLC_Functional_Test_11 AND NOT #Aux_Trigger_11;   // rising edge of #In_Functional_Test_Odd.Star_Test_PLC_Functional_Test_11
   #Aux_Trigger_11 := #In_Functional_Test_Odd.Star_Test_PLC_Functional_Test_11;
   IF #_w1 THEN
       #Functional_Tests_Panels[11].Water_Fountain := #Water_Fountain;
       #Functional_Tests_Panels[11].Serial_Number := #Serial_Number;
   END_IF;
   IF #In_Functional_Test_Odd.Star_Test_PLC_Functional_Test_11 THEN
       #Functional_Tests_Panels[11].Read_Electrical_Voltage := #Read_Electrial_Voltage;
   END_IF;
   IF #In_Functional_Test_Odd.Star_Test_PLC_Functional_Test_11 AND NOT #In_Functional_Test_Odd.Electrical_Current_Test_Approved_PLC_Functional_Test_11 THEN
       #Functional_Tests_Panels[11].Electrical_Current_Test := 'REPROVADO';
       #Functional_Tests_Panels[11].Read_Electrical_Current := #In_Functional_Test_Odd.Electrical_Current_Read_PLC_Functional_Test_11;
   END_IF;
   IF #In_Functional_Test_Odd.Star_Test_PLC_Functional_Test_11 AND #In_Functional_Test_Odd.Electrical_Current_Test_Approved_PLC_Functional_Test_11 THEN
       #Functional_Tests_Panels[11].Electrical_Current_Test := 'APROVADO';
   END_IF;
   IF #In_Functional_Test_Odd.Star_Test_PLC_Functional_Test_11 AND #In_Functional_Test_Odd.Visual_Test_Approved_PLC_Functional_Test_11 THEN
       #Functional_Tests_Panels[11].Visual_Test := 'APROVADO';
   END_IF;
   IF #In_Functional_Test_Odd.Star_Test_PLC_Functional_Test_11 AND NOT #In_Functional_Test_Odd.Visual_Test_Approved_PLC_Functional_Test_11 THEN
       #Functional_Tests_Panels[11].Visual_Test := 'REPROVADO';
   END_IF;
   IF #In_Functional_Test_Odd.Star_Test_PLC_Functional_Test_11 AND #In_Functional_Test_Odd.Electrical_Current_Test_Approved_PLC_Functional_Test_11 AND #In_Functional_Test_Odd.Visual_Test_Approved_PLC_Functional_Test_11 THEN
       #Functional_Tests_Panels[11].Functional_Test := 'APROVADO';
   END_IF;
   IF #In_Functional_Test_Odd.Star_Test_PLC_Functional_Test_11 AND (NOT #In_Functional_Test_Odd.Electrical_Current_Test_Approved_PLC_Functional_Test_11 OR NOT #In_Functional_Test_Odd.Visual_Test_Approved_PLC_Functional_Test_11) THEN
       #Functional_Tests_Panels[11].Functional_Test := 'REPROVADO';
   END_IF;
END_REGION

REGION Network 12: Panel 12
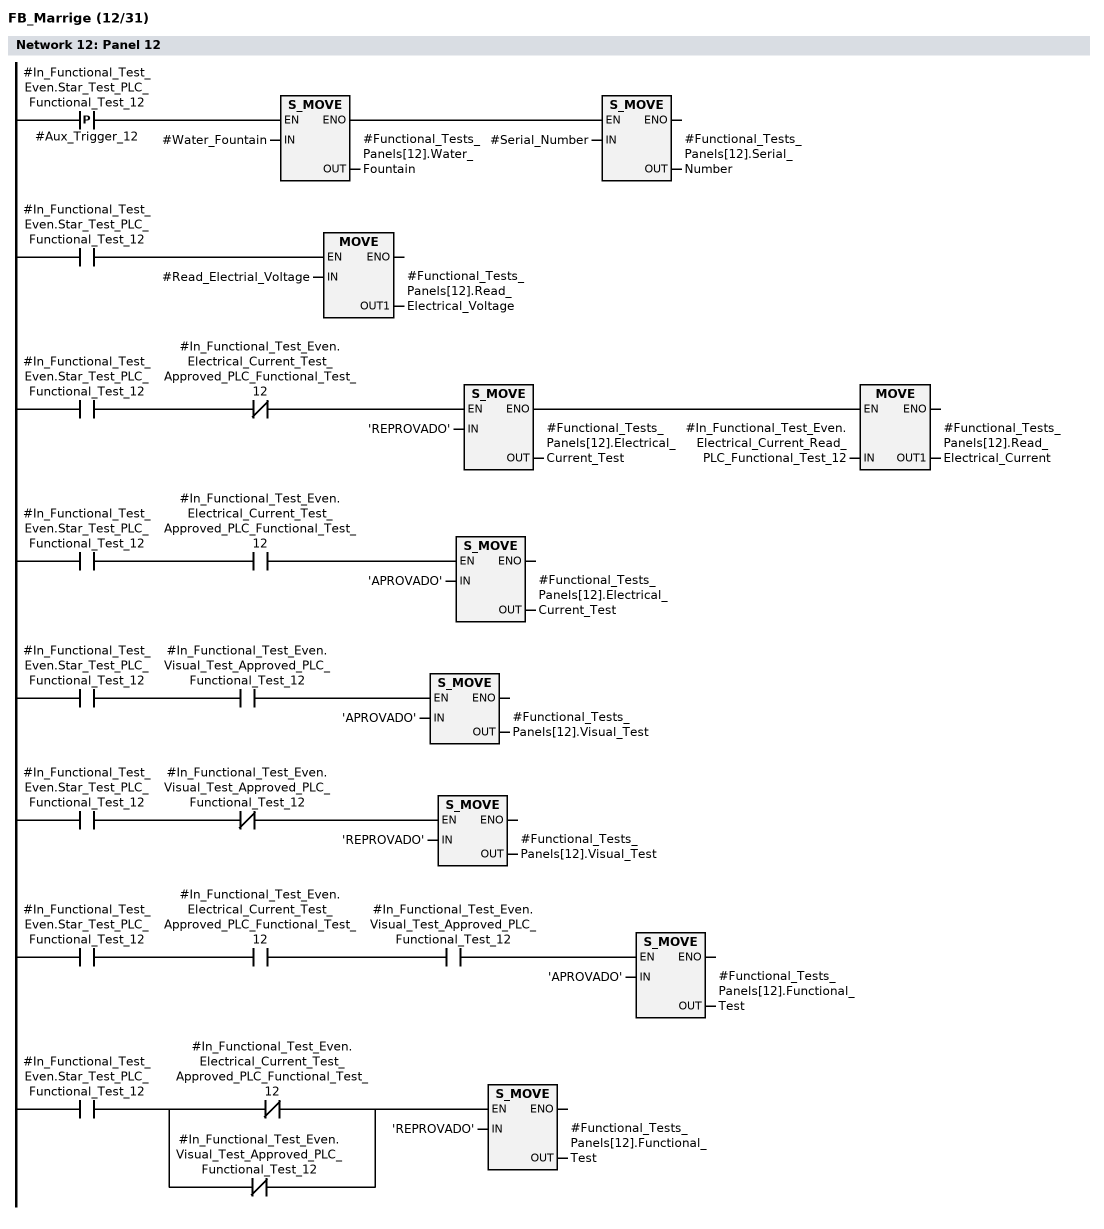
   RUNG wire#powerrail
      P_Contact(operand := #In_Functional_Test_Even.Star_Test_PLC_Functional_Test_12, bit := #Aux_Trigger_12)
      S_Move(in := #Water_Fountain, out => #Functional_Tests_Panels[12].Water_Fountain)
      S_Move(in := #Serial_Number, out => #Functional_Tests_Panels[12].Serial_Number)
   END_RUNG
   RUNG wire#powerrail
      Contact( #In_Functional_Test_Even.Star_Test_PLC_Functional_Test_12 )
      Move(in := #Read_Electrial_Voltage, out1 => #Functional_Tests_Panels[12].Read_Electrical_Voltage)
   END_RUNG
   RUNG wire#powerrail
      Contact( #In_Functional_Test_Even.Star_Test_PLC_Functional_Test_12 )
      I_Contact( #In_Functional_Test_Even.Electrical_Current_Test_Approved_PLC_Functional_Test_12 )
      S_Move(in := 'REPROVADO', out => #Functional_Tests_Panels[12].Electrical_Current_Test)
      Move(in := #In_Functional_Test_Even.Electrical_Current_Read_PLC_Functional_Test_12, out1 => #Functional_Tests_Panels[12].Read_Electrical_Current)
   END_RUNG
   RUNG wire#powerrail
      Contact( #In_Functional_Test_Even.Star_Test_PLC_Functional_Test_12 )
      Contact( #In_Functional_Test_Even.Electrical_Current_Test_Approved_PLC_Functional_Test_12 )
      S_Move(in := 'APROVADO', out => #Functional_Tests_Panels[12].Electrical_Current_Test)
   END_RUNG
   RUNG wire#powerrail
      Contact( #In_Functional_Test_Even.Star_Test_PLC_Functional_Test_12 )
      Contact( #In_Functional_Test_Even.Visual_Test_Approved_PLC_Functional_Test_12 )
      S_Move(in := 'APROVADO', out => #Functional_Tests_Panels[12].Visual_Test)
   END_RUNG
   RUNG wire#powerrail
      Contact( #In_Functional_Test_Even.Star_Test_PLC_Functional_Test_12 )
      I_Contact( #In_Functional_Test_Even.Visual_Test_Approved_PLC_Functional_Test_12 )
      S_Move(in := 'REPROVADO', out => #Functional_Tests_Panels[12].Visual_Test)
   END_RUNG
   RUNG wire#powerrail
      Contact( #In_Functional_Test_Even.Star_Test_PLC_Functional_Test_12 )
      Contact( #In_Functional_Test_Even.Electrical_Current_Test_Approved_PLC_Functional_Test_12 )
      Contact( #In_Functional_Test_Even.Visual_Test_Approved_PLC_Functional_Test_12 )
      S_Move(in := 'APROVADO', out => #Functional_Tests_Panels[12].Functional_Test)
   END_RUNG
   RUNG wire#powerrail
      Contact( #In_Functional_Test_Even.Star_Test_PLC_Functional_Test_12 )
      wire#w1
      I_Contact( #In_Functional_Test_Even.Electrical_Current_Test_Approved_PLC_Functional_Test_12 )
      wire#w2
      S_Move(in := 'REPROVADO', out => #Functional_Tests_Panels[12].Functional_Test)
   END_RUNG
   RUNG wire#w1
      I_Contact( #In_Functional_Test_Even.Visual_Test_Approved_PLC_Functional_Test_12 )
   END_RUNG wire#w2
   // the same network as SCL:
   #_w1 := #In_Functional_Test_Even.Star_Test_PLC_Functional_Test_12 AND NOT #Aux_Trigger_12;   // rising edge of #In_Functional_Test_Even.Star_Test_PLC_Functional_Test_12
   #Aux_Trigger_12 := #In_Functional_Test_Even.Star_Test_PLC_Functional_Test_12;
   IF #_w1 THEN
       #Functional_Tests_Panels[12].Water_Fountain := #Water_Fountain;
       #Functional_Tests_Panels[12].Serial_Number := #Serial_Number;
   END_IF;
   IF #In_Functional_Test_Even.Star_Test_PLC_Functional_Test_12 THEN
       #Functional_Tests_Panels[12].Read_Electrical_Voltage := #Read_Electrial_Voltage;
   END_IF;
   IF #In_Functional_Test_Even.Star_Test_PLC_Functional_Test_12 AND NOT #In_Functional_Test_Even.Electrical_Current_Test_Approved_PLC_Functional_Test_12 THEN
       #Functional_Tests_Panels[12].Electrical_Current_Test := 'REPROVADO';
       #Functional_Tests_Panels[12].Read_Electrical_Current := #In_Functional_Test_Even.Electrical_Current_Read_PLC_Functional_Test_12;
   END_IF;
   IF #In_Functional_Test_Even.Star_Test_PLC_Functional_Test_12 AND #In_Functional_Test_Even.Electrical_Current_Test_Approved_PLC_Functional_Test_12 THEN
       #Functional_Tests_Panels[12].Electrical_Current_Test := 'APROVADO';
   END_IF;
   IF #In_Functional_Test_Even.Star_Test_PLC_Functional_Test_12 AND #In_Functional_Test_Even.Visual_Test_Approved_PLC_Functional_Test_12 THEN
       #Functional_Tests_Panels[12].Visual_Test := 'APROVADO';
   END_IF;
   IF #In_Functional_Test_Even.Star_Test_PLC_Functional_Test_12 AND NOT #In_Functional_Test_Even.Visual_Test_Approved_PLC_Functional_Test_12 THEN
       #Functional_Tests_Panels[12].Visual_Test := 'REPROVADO';
   END_IF;
   IF #In_Functional_Test_Even.Star_Test_PLC_Functional_Test_12 AND #In_Functional_Test_Even.Electrical_Current_Test_Approved_PLC_Functional_Test_12 AND #In_Functional_Test_Even.Visual_Test_Approved_PLC_Functional_Test_12 THEN
       #Functional_Tests_Panels[12].Functional_Test := 'APROVADO';
   END_IF;
   IF #In_Functional_Test_Even.Star_Test_PLC_Functional_Test_12 AND (NOT #In_Functional_Test_Even.Electrical_Current_Test_Approved_PLC_Functional_Test_12 OR NOT #In_Functional_Test_Even.Visual_Test_Approved_PLC_Functional_Test_12) THEN
       #Functional_Tests_Panels[12].Functional_Test := 'REPROVADO';
   END_IF;
END_REGION

REGION Network 13: Panel 13
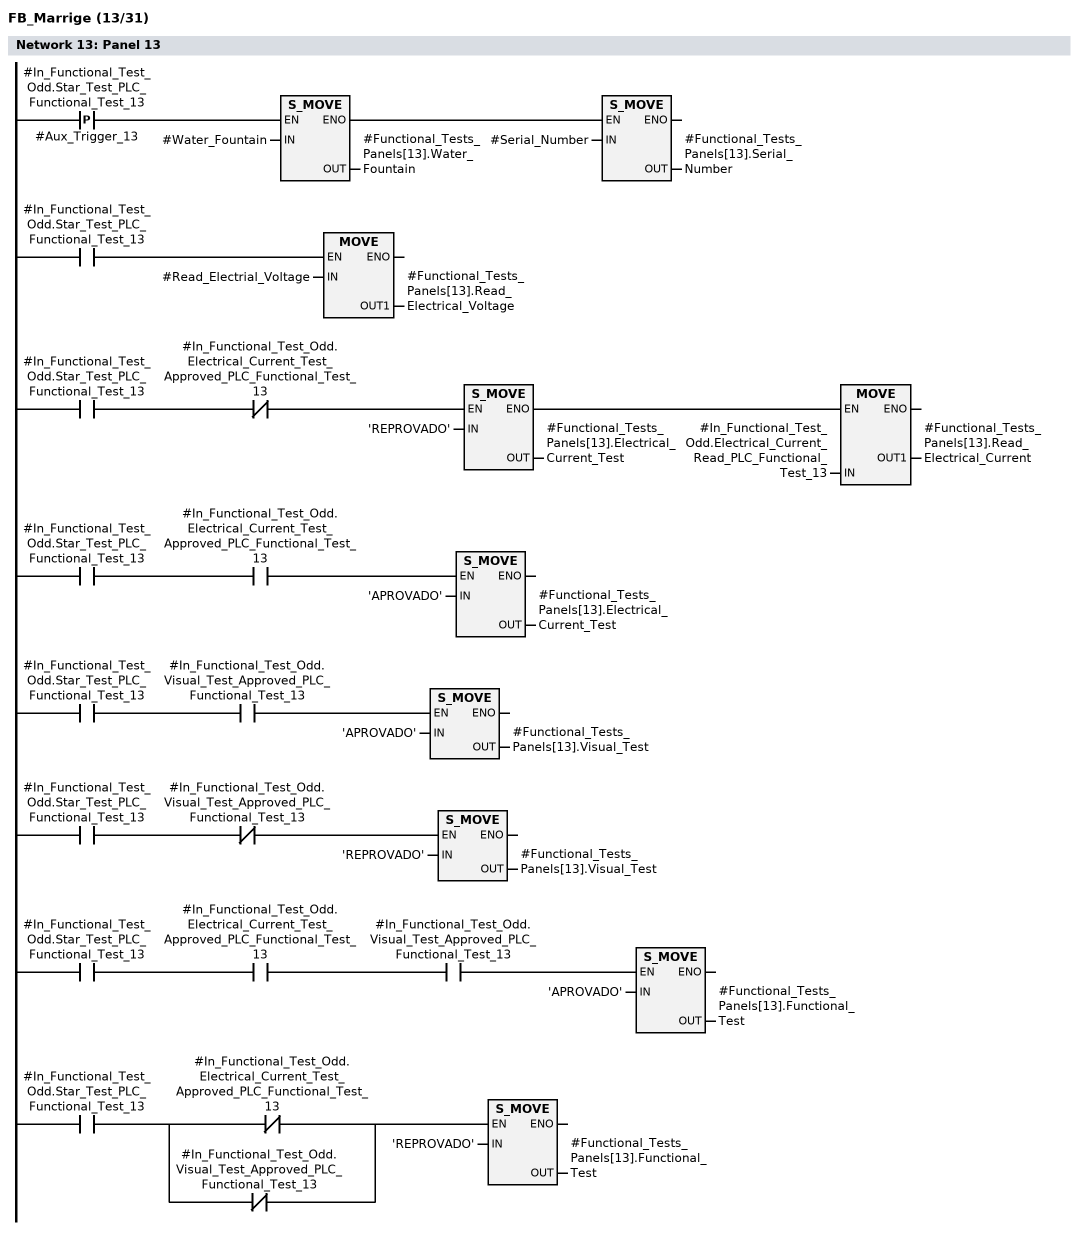
   RUNG wire#powerrail
      P_Contact(operand := #In_Functional_Test_Odd.Star_Test_PLC_Functional_Test_13, bit := #Aux_Trigger_13)
      S_Move(in := #Water_Fountain, out => #Functional_Tests_Panels[13].Water_Fountain)
      S_Move(in := #Serial_Number, out => #Functional_Tests_Panels[13].Serial_Number)
   END_RUNG
   RUNG wire#powerrail
      Contact( #In_Functional_Test_Odd.Star_Test_PLC_Functional_Test_13 )
      Move(in := #Read_Electrial_Voltage, out1 => #Functional_Tests_Panels[13].Read_Electrical_Voltage)
   END_RUNG
   RUNG wire#powerrail
      Contact( #In_Functional_Test_Odd.Star_Test_PLC_Functional_Test_13 )
      I_Contact( #In_Functional_Test_Odd.Electrical_Current_Test_Approved_PLC_Functional_Test_13 )
      S_Move(in := 'REPROVADO', out => #Functional_Tests_Panels[13].Electrical_Current_Test)
      Move(in := #In_Functional_Test_Odd.Electrical_Current_Read_PLC_Functional_Test_13, out1 => #Functional_Tests_Panels[13].Read_Electrical_Current)
   END_RUNG
   RUNG wire#powerrail
      Contact( #In_Functional_Test_Odd.Star_Test_PLC_Functional_Test_13 )
      Contact( #In_Functional_Test_Odd.Electrical_Current_Test_Approved_PLC_Functional_Test_13 )
      S_Move(in := 'APROVADO', out => #Functional_Tests_Panels[13].Electrical_Current_Test)
   END_RUNG
   RUNG wire#powerrail
      Contact( #In_Functional_Test_Odd.Star_Test_PLC_Functional_Test_13 )
      Contact( #In_Functional_Test_Odd.Visual_Test_Approved_PLC_Functional_Test_13 )
      S_Move(in := 'APROVADO', out => #Functional_Tests_Panels[13].Visual_Test)
   END_RUNG
   RUNG wire#powerrail
      Contact( #In_Functional_Test_Odd.Star_Test_PLC_Functional_Test_13 )
      I_Contact( #In_Functional_Test_Odd.Visual_Test_Approved_PLC_Functional_Test_13 )
      S_Move(in := 'REPROVADO', out => #Functional_Tests_Panels[13].Visual_Test)
   END_RUNG
   RUNG wire#powerrail
      Contact( #In_Functional_Test_Odd.Star_Test_PLC_Functional_Test_13 )
      Contact( #In_Functional_Test_Odd.Electrical_Current_Test_Approved_PLC_Functional_Test_13 )
      Contact( #In_Functional_Test_Odd.Visual_Test_Approved_PLC_Functional_Test_13 )
      S_Move(in := 'APROVADO', out => #Functional_Tests_Panels[13].Functional_Test)
   END_RUNG
   RUNG wire#powerrail
      Contact( #In_Functional_Test_Odd.Star_Test_PLC_Functional_Test_13 )
      wire#w1
      I_Contact( #In_Functional_Test_Odd.Electrical_Current_Test_Approved_PLC_Functional_Test_13 )
      wire#w2
      S_Move(in := 'REPROVADO', out => #Functional_Tests_Panels[13].Functional_Test)
   END_RUNG
   RUNG wire#w1
      I_Contact( #In_Functional_Test_Odd.Visual_Test_Approved_PLC_Functional_Test_13 )
   END_RUNG wire#w2
   // the same network as SCL:
   #_w1 := #In_Functional_Test_Odd.Star_Test_PLC_Functional_Test_13 AND NOT #Aux_Trigger_13;   // rising edge of #In_Functional_Test_Odd.Star_Test_PLC_Functional_Test_13
   #Aux_Trigger_13 := #In_Functional_Test_Odd.Star_Test_PLC_Functional_Test_13;
   IF #_w1 THEN
       #Functional_Tests_Panels[13].Water_Fountain := #Water_Fountain;
       #Functional_Tests_Panels[13].Serial_Number := #Serial_Number;
   END_IF;
   IF #In_Functional_Test_Odd.Star_Test_PLC_Functional_Test_13 THEN
       #Functional_Tests_Panels[13].Read_Electrical_Voltage := #Read_Electrial_Voltage;
   END_IF;
   IF #In_Functional_Test_Odd.Star_Test_PLC_Functional_Test_13 AND NOT #In_Functional_Test_Odd.Electrical_Current_Test_Approved_PLC_Functional_Test_13 THEN
       #Functional_Tests_Panels[13].Electrical_Current_Test := 'REPROVADO';
       #Functional_Tests_Panels[13].Read_Electrical_Current := #In_Functional_Test_Odd.Electrical_Current_Read_PLC_Functional_Test_13;
   END_IF;
   IF #In_Functional_Test_Odd.Star_Test_PLC_Functional_Test_13 AND #In_Functional_Test_Odd.Electrical_Current_Test_Approved_PLC_Functional_Test_13 THEN
       #Functional_Tests_Panels[13].Electrical_Current_Test := 'APROVADO';
   END_IF;
   IF #In_Functional_Test_Odd.Star_Test_PLC_Functional_Test_13 AND #In_Functional_Test_Odd.Visual_Test_Approved_PLC_Functional_Test_13 THEN
       #Functional_Tests_Panels[13].Visual_Test := 'APROVADO';
   END_IF;
   IF #In_Functional_Test_Odd.Star_Test_PLC_Functional_Test_13 AND NOT #In_Functional_Test_Odd.Visual_Test_Approved_PLC_Functional_Test_13 THEN
       #Functional_Tests_Panels[13].Visual_Test := 'REPROVADO';
   END_IF;
   IF #In_Functional_Test_Odd.Star_Test_PLC_Functional_Test_13 AND #In_Functional_Test_Odd.Electrical_Current_Test_Approved_PLC_Functional_Test_13 AND #In_Functional_Test_Odd.Visual_Test_Approved_PLC_Functional_Test_13 THEN
       #Functional_Tests_Panels[13].Functional_Test := 'APROVADO';
   END_IF;
   IF #In_Functional_Test_Odd.Star_Test_PLC_Functional_Test_13 AND (NOT #In_Functional_Test_Odd.Electrical_Current_Test_Approved_PLC_Functional_Test_13 OR NOT #In_Functional_Test_Odd.Visual_Test_Approved_PLC_Functional_Test_13) THEN
       #Functional_Tests_Panels[13].Functional_Test := 'REPROVADO';
   END_IF;
END_REGION

REGION Network 14: Panel 14
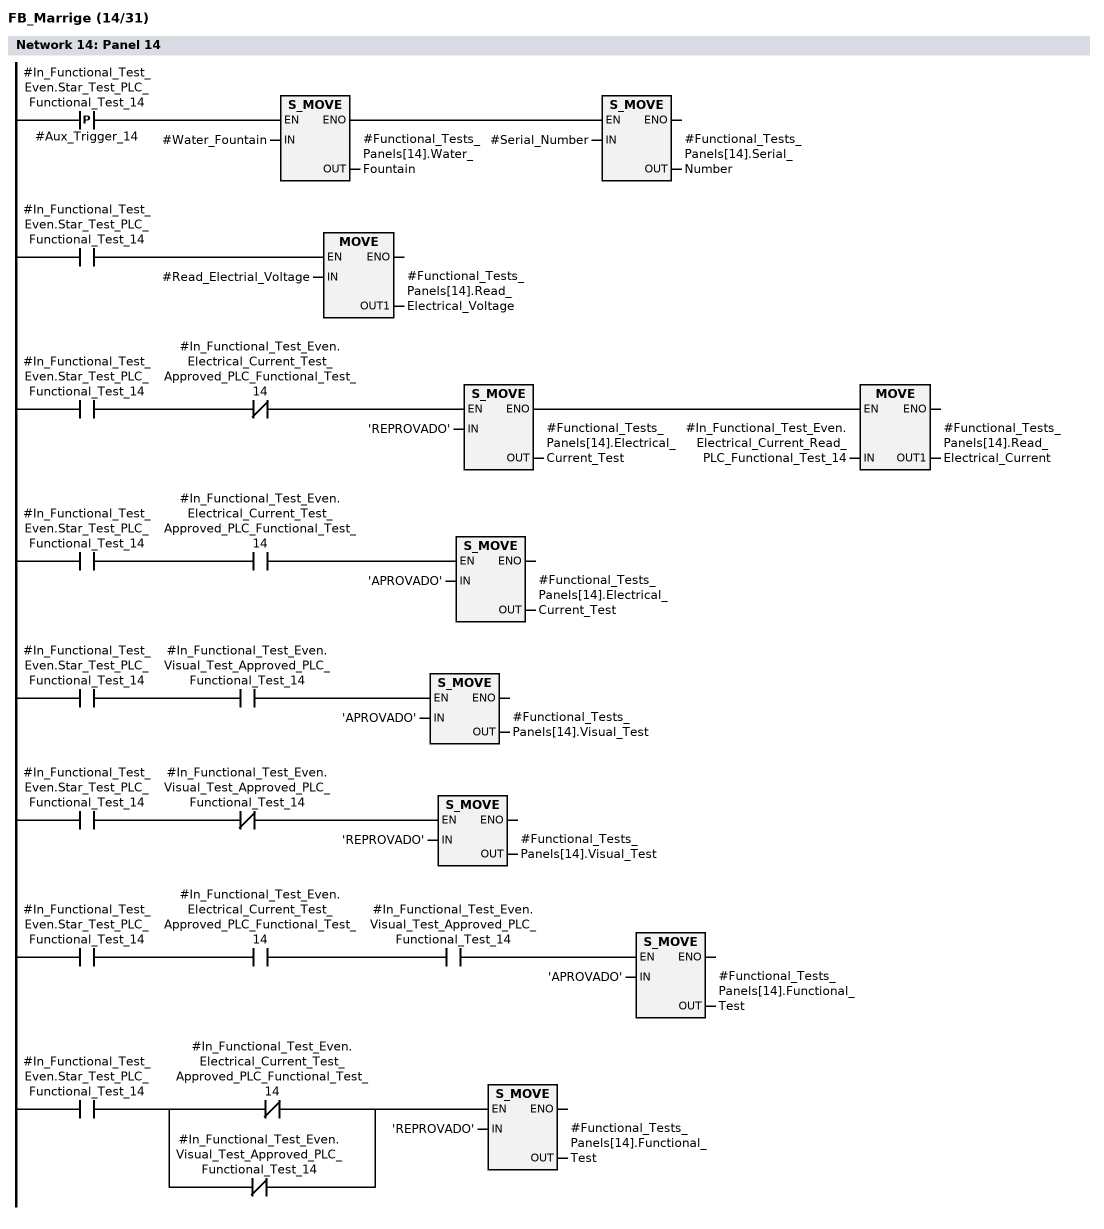
   RUNG wire#powerrail
      P_Contact(operand := #In_Functional_Test_Even.Star_Test_PLC_Functional_Test_14, bit := #Aux_Trigger_14)
      S_Move(in := #Water_Fountain, out => #Functional_Tests_Panels[14].Water_Fountain)
      S_Move(in := #Serial_Number, out => #Functional_Tests_Panels[14].Serial_Number)
   END_RUNG
   RUNG wire#powerrail
      Contact( #In_Functional_Test_Even.Star_Test_PLC_Functional_Test_14 )
      Move(in := #Read_Electrial_Voltage, out1 => #Functional_Tests_Panels[14].Read_Electrical_Voltage)
   END_RUNG
   RUNG wire#powerrail
      Contact( #In_Functional_Test_Even.Star_Test_PLC_Functional_Test_14 )
      I_Contact( #In_Functional_Test_Even.Electrical_Current_Test_Approved_PLC_Functional_Test_14 )
      S_Move(in := 'REPROVADO', out => #Functional_Tests_Panels[14].Electrical_Current_Test)
      Move(in := #In_Functional_Test_Even.Electrical_Current_Read_PLC_Functional_Test_14, out1 => #Functional_Tests_Panels[14].Read_Electrical_Current)
   END_RUNG
   RUNG wire#powerrail
      Contact( #In_Functional_Test_Even.Star_Test_PLC_Functional_Test_14 )
      Contact( #In_Functional_Test_Even.Electrical_Current_Test_Approved_PLC_Functional_Test_14 )
      S_Move(in := 'APROVADO', out => #Functional_Tests_Panels[14].Electrical_Current_Test)
   END_RUNG
   RUNG wire#powerrail
      Contact( #In_Functional_Test_Even.Star_Test_PLC_Functional_Test_14 )
      Contact( #In_Functional_Test_Even.Visual_Test_Approved_PLC_Functional_Test_14 )
      S_Move(in := 'APROVADO', out => #Functional_Tests_Panels[14].Visual_Test)
   END_RUNG
   RUNG wire#powerrail
      Contact( #In_Functional_Test_Even.Star_Test_PLC_Functional_Test_14 )
      I_Contact( #In_Functional_Test_Even.Visual_Test_Approved_PLC_Functional_Test_14 )
      S_Move(in := 'REPROVADO', out => #Functional_Tests_Panels[14].Visual_Test)
   END_RUNG
   RUNG wire#powerrail
      Contact( #In_Functional_Test_Even.Star_Test_PLC_Functional_Test_14 )
      Contact( #In_Functional_Test_Even.Electrical_Current_Test_Approved_PLC_Functional_Test_14 )
      Contact( #In_Functional_Test_Even.Visual_Test_Approved_PLC_Functional_Test_14 )
      S_Move(in := 'APROVADO', out => #Functional_Tests_Panels[14].Functional_Test)
   END_RUNG
   RUNG wire#powerrail
      Contact( #In_Functional_Test_Even.Star_Test_PLC_Functional_Test_14 )
      wire#w1
      I_Contact( #In_Functional_Test_Even.Electrical_Current_Test_Approved_PLC_Functional_Test_14 )
      wire#w2
      S_Move(in := 'REPROVADO', out => #Functional_Tests_Panels[14].Functional_Test)
   END_RUNG
   RUNG wire#w1
      I_Contact( #In_Functional_Test_Even.Visual_Test_Approved_PLC_Functional_Test_14 )
   END_RUNG wire#w2
   // the same network as SCL:
   #_w1 := #In_Functional_Test_Even.Star_Test_PLC_Functional_Test_14 AND NOT #Aux_Trigger_14;   // rising edge of #In_Functional_Test_Even.Star_Test_PLC_Functional_Test_14
   #Aux_Trigger_14 := #In_Functional_Test_Even.Star_Test_PLC_Functional_Test_14;
   IF #_w1 THEN
       #Functional_Tests_Panels[14].Water_Fountain := #Water_Fountain;
       #Functional_Tests_Panels[14].Serial_Number := #Serial_Number;
   END_IF;
   IF #In_Functional_Test_Even.Star_Test_PLC_Functional_Test_14 THEN
       #Functional_Tests_Panels[14].Read_Electrical_Voltage := #Read_Electrial_Voltage;
   END_IF;
   IF #In_Functional_Test_Even.Star_Test_PLC_Functional_Test_14 AND NOT #In_Functional_Test_Even.Electrical_Current_Test_Approved_PLC_Functional_Test_14 THEN
       #Functional_Tests_Panels[14].Electrical_Current_Test := 'REPROVADO';
       #Functional_Tests_Panels[14].Read_Electrical_Current := #In_Functional_Test_Even.Electrical_Current_Read_PLC_Functional_Test_14;
   END_IF;
   IF #In_Functional_Test_Even.Star_Test_PLC_Functional_Test_14 AND #In_Functional_Test_Even.Electrical_Current_Test_Approved_PLC_Functional_Test_14 THEN
       #Functional_Tests_Panels[14].Electrical_Current_Test := 'APROVADO';
   END_IF;
   IF #In_Functional_Test_Even.Star_Test_PLC_Functional_Test_14 AND #In_Functional_Test_Even.Visual_Test_Approved_PLC_Functional_Test_14 THEN
       #Functional_Tests_Panels[14].Visual_Test := 'APROVADO';
   END_IF;
   IF #In_Functional_Test_Even.Star_Test_PLC_Functional_Test_14 AND NOT #In_Functional_Test_Even.Visual_Test_Approved_PLC_Functional_Test_14 THEN
       #Functional_Tests_Panels[14].Visual_Test := 'REPROVADO';
   END_IF;
   IF #In_Functional_Test_Even.Star_Test_PLC_Functional_Test_14 AND #In_Functional_Test_Even.Electrical_Current_Test_Approved_PLC_Functional_Test_14 AND #In_Functional_Test_Even.Visual_Test_Approved_PLC_Functional_Test_14 THEN
       #Functional_Tests_Panels[14].Functional_Test := 'APROVADO';
   END_IF;
   IF #In_Functional_Test_Even.Star_Test_PLC_Functional_Test_14 AND (NOT #In_Functional_Test_Even.Electrical_Current_Test_Approved_PLC_Functional_Test_14 OR NOT #In_Functional_Test_Even.Visual_Test_Approved_PLC_Functional_Test_14) THEN
       #Functional_Tests_Panels[14].Functional_Test := 'REPROVADO';
   END_IF;
END_REGION

REGION Network 15: Panel 15
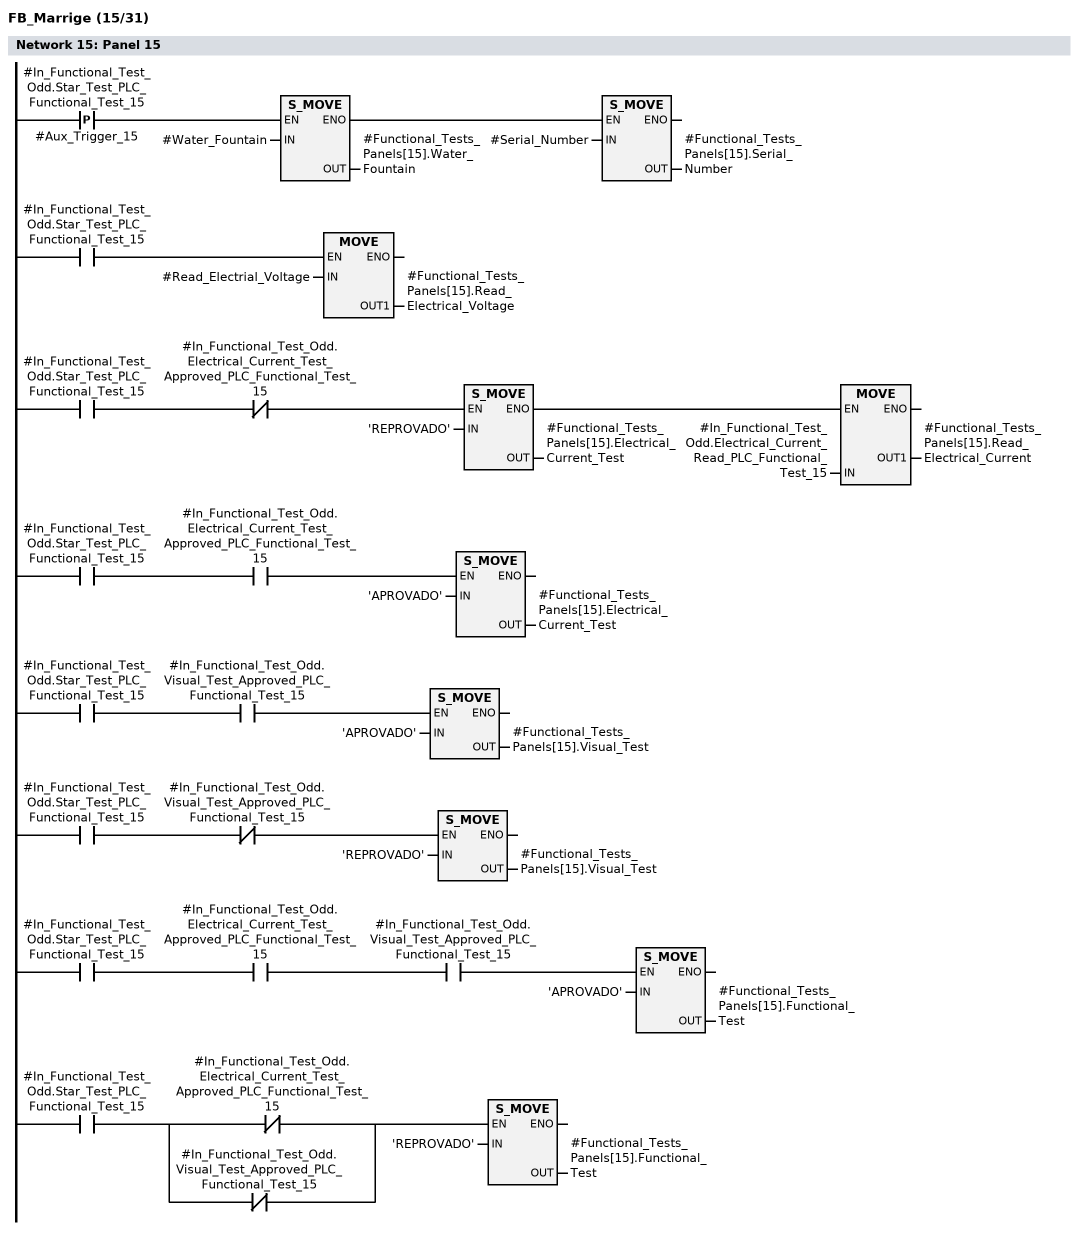
   RUNG wire#powerrail
      P_Contact(operand := #In_Functional_Test_Odd.Star_Test_PLC_Functional_Test_15, bit := #Aux_Trigger_15)
      S_Move(in := #Water_Fountain, out => #Functional_Tests_Panels[15].Water_Fountain)
      S_Move(in := #Serial_Number, out => #Functional_Tests_Panels[15].Serial_Number)
   END_RUNG
   RUNG wire#powerrail
      Contact( #In_Functional_Test_Odd.Star_Test_PLC_Functional_Test_15 )
      Move(in := #Read_Electrial_Voltage, out1 => #Functional_Tests_Panels[15].Read_Electrical_Voltage)
   END_RUNG
   RUNG wire#powerrail
      Contact( #In_Functional_Test_Odd.Star_Test_PLC_Functional_Test_15 )
      I_Contact( #In_Functional_Test_Odd.Electrical_Current_Test_Approved_PLC_Functional_Test_15 )
      S_Move(in := 'REPROVADO', out => #Functional_Tests_Panels[15].Electrical_Current_Test)
      Move(in := #In_Functional_Test_Odd.Electrical_Current_Read_PLC_Functional_Test_15, out1 => #Functional_Tests_Panels[15].Read_Electrical_Current)
   END_RUNG
   RUNG wire#powerrail
      Contact( #In_Functional_Test_Odd.Star_Test_PLC_Functional_Test_15 )
      Contact( #In_Functional_Test_Odd.Electrical_Current_Test_Approved_PLC_Functional_Test_15 )
      S_Move(in := 'APROVADO', out => #Functional_Tests_Panels[15].Electrical_Current_Test)
   END_RUNG
   RUNG wire#powerrail
      Contact( #In_Functional_Test_Odd.Star_Test_PLC_Functional_Test_15 )
      Contact( #In_Functional_Test_Odd.Visual_Test_Approved_PLC_Functional_Test_15 )
      S_Move(in := 'APROVADO', out => #Functional_Tests_Panels[15].Visual_Test)
   END_RUNG
   RUNG wire#powerrail
      Contact( #In_Functional_Test_Odd.Star_Test_PLC_Functional_Test_15 )
      I_Contact( #In_Functional_Test_Odd.Visual_Test_Approved_PLC_Functional_Test_15 )
      S_Move(in := 'REPROVADO', out => #Functional_Tests_Panels[15].Visual_Test)
   END_RUNG
   RUNG wire#powerrail
      Contact( #In_Functional_Test_Odd.Star_Test_PLC_Functional_Test_15 )
      Contact( #In_Functional_Test_Odd.Electrical_Current_Test_Approved_PLC_Functional_Test_15 )
      Contact( #In_Functional_Test_Odd.Visual_Test_Approved_PLC_Functional_Test_15 )
      S_Move(in := 'APROVADO', out => #Functional_Tests_Panels[15].Functional_Test)
   END_RUNG
   RUNG wire#powerrail
      Contact( #In_Functional_Test_Odd.Star_Test_PLC_Functional_Test_15 )
      wire#w1
      I_Contact( #In_Functional_Test_Odd.Electrical_Current_Test_Approved_PLC_Functional_Test_15 )
      wire#w2
      S_Move(in := 'REPROVADO', out => #Functional_Tests_Panels[15].Functional_Test)
   END_RUNG
   RUNG wire#w1
      I_Contact( #In_Functional_Test_Odd.Visual_Test_Approved_PLC_Functional_Test_15 )
   END_RUNG wire#w2
   // the same network as SCL:
   #_w1 := #In_Functional_Test_Odd.Star_Test_PLC_Functional_Test_15 AND NOT #Aux_Trigger_15;   // rising edge of #In_Functional_Test_Odd.Star_Test_PLC_Functional_Test_15
   #Aux_Trigger_15 := #In_Functional_Test_Odd.Star_Test_PLC_Functional_Test_15;
   IF #_w1 THEN
       #Functional_Tests_Panels[15].Water_Fountain := #Water_Fountain;
       #Functional_Tests_Panels[15].Serial_Number := #Serial_Number;
   END_IF;
   IF #In_Functional_Test_Odd.Star_Test_PLC_Functional_Test_15 THEN
       #Functional_Tests_Panels[15].Read_Electrical_Voltage := #Read_Electrial_Voltage;
   END_IF;
   IF #In_Functional_Test_Odd.Star_Test_PLC_Functional_Test_15 AND NOT #In_Functional_Test_Odd.Electrical_Current_Test_Approved_PLC_Functional_Test_15 THEN
       #Functional_Tests_Panels[15].Electrical_Current_Test := 'REPROVADO';
       #Functional_Tests_Panels[15].Read_Electrical_Current := #In_Functional_Test_Odd.Electrical_Current_Read_PLC_Functional_Test_15;
   END_IF;
   IF #In_Functional_Test_Odd.Star_Test_PLC_Functional_Test_15 AND #In_Functional_Test_Odd.Electrical_Current_Test_Approved_PLC_Functional_Test_15 THEN
       #Functional_Tests_Panels[15].Electrical_Current_Test := 'APROVADO';
   END_IF;
   IF #In_Functional_Test_Odd.Star_Test_PLC_Functional_Test_15 AND #In_Functional_Test_Odd.Visual_Test_Approved_PLC_Functional_Test_15 THEN
       #Functional_Tests_Panels[15].Visual_Test := 'APROVADO';
   END_IF;
   IF #In_Functional_Test_Odd.Star_Test_PLC_Functional_Test_15 AND NOT #In_Functional_Test_Odd.Visual_Test_Approved_PLC_Functional_Test_15 THEN
       #Functional_Tests_Panels[15].Visual_Test := 'REPROVADO';
   END_IF;
   IF #In_Functional_Test_Odd.Star_Test_PLC_Functional_Test_15 AND #In_Functional_Test_Odd.Electrical_Current_Test_Approved_PLC_Functional_Test_15 AND #In_Functional_Test_Odd.Visual_Test_Approved_PLC_Functional_Test_15 THEN
       #Functional_Tests_Panels[15].Functional_Test := 'APROVADO';
   END_IF;
   IF #In_Functional_Test_Odd.Star_Test_PLC_Functional_Test_15 AND (NOT #In_Functional_Test_Odd.Electrical_Current_Test_Approved_PLC_Functional_Test_15 OR NOT #In_Functional_Test_Odd.Visual_Test_Approved_PLC_Functional_Test_15) THEN
       #Functional_Tests_Panels[15].Functional_Test := 'REPROVADO';
   END_IF;
END_REGION

REGION Network 16: Panel 16
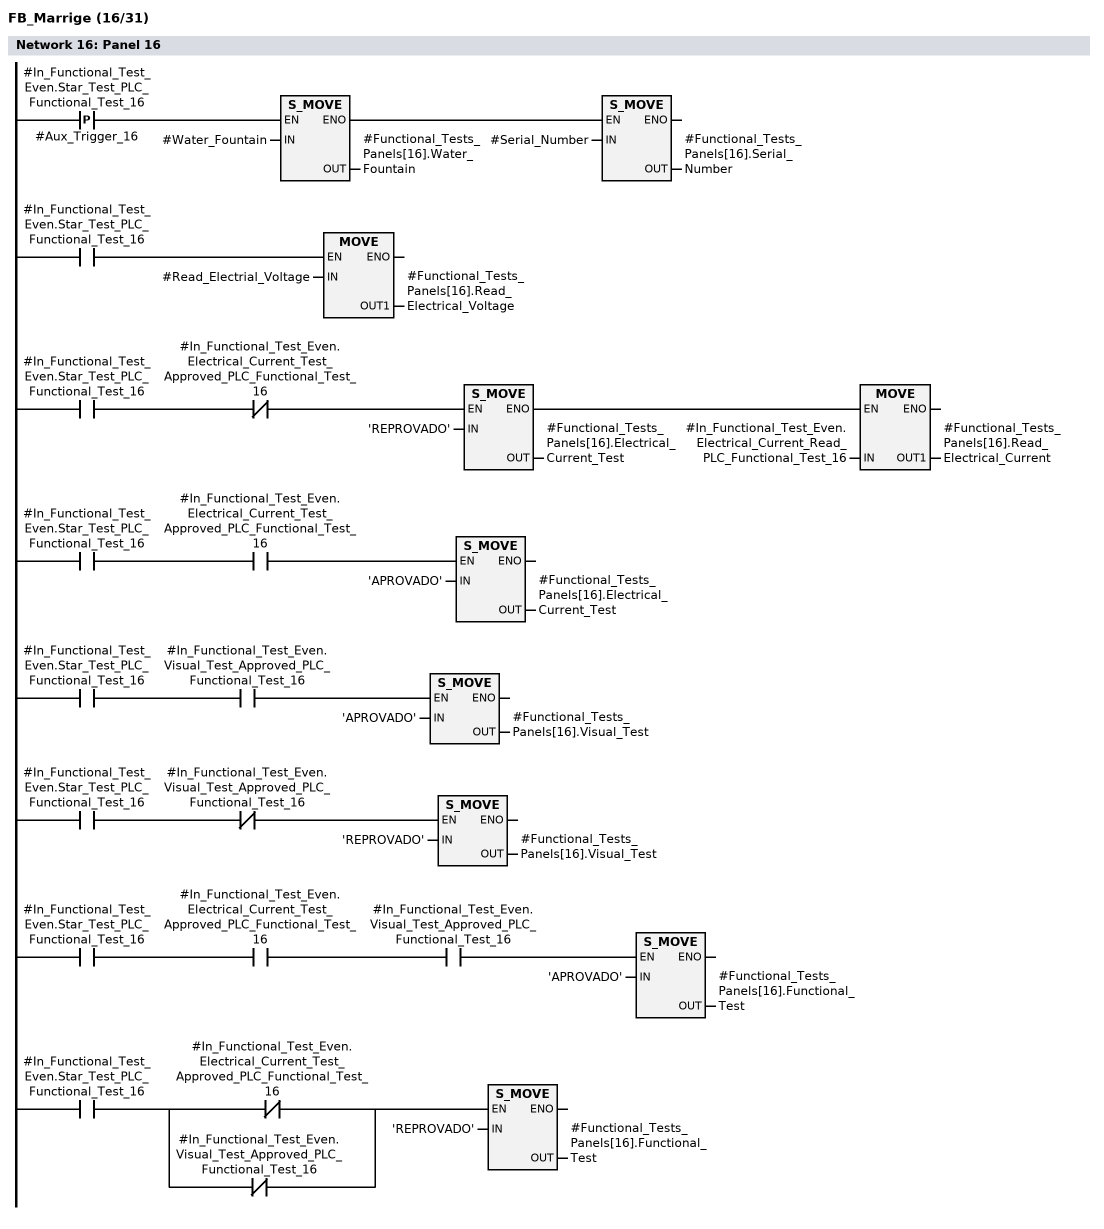
   RUNG wire#powerrail
      P_Contact(operand := #In_Functional_Test_Even.Star_Test_PLC_Functional_Test_16, bit := #Aux_Trigger_16)
      S_Move(in := #Water_Fountain, out => #Functional_Tests_Panels[16].Water_Fountain)
      S_Move(in := #Serial_Number, out => #Functional_Tests_Panels[16].Serial_Number)
   END_RUNG
   RUNG wire#powerrail
      Contact( #In_Functional_Test_Even.Star_Test_PLC_Functional_Test_16 )
      Move(in := #Read_Electrial_Voltage, out1 => #Functional_Tests_Panels[16].Read_Electrical_Voltage)
   END_RUNG
   RUNG wire#powerrail
      Contact( #In_Functional_Test_Even.Star_Test_PLC_Functional_Test_16 )
      I_Contact( #In_Functional_Test_Even.Electrical_Current_Test_Approved_PLC_Functional_Test_16 )
      S_Move(in := 'REPROVADO', out => #Functional_Tests_Panels[16].Electrical_Current_Test)
      Move(in := #In_Functional_Test_Even.Electrical_Current_Read_PLC_Functional_Test_16, out1 => #Functional_Tests_Panels[16].Read_Electrical_Current)
   END_RUNG
   RUNG wire#powerrail
      Contact( #In_Functional_Test_Even.Star_Test_PLC_Functional_Test_16 )
      Contact( #In_Functional_Test_Even.Electrical_Current_Test_Approved_PLC_Functional_Test_16 )
      S_Move(in := 'APROVADO', out => #Functional_Tests_Panels[16].Electrical_Current_Test)
   END_RUNG
   RUNG wire#powerrail
      Contact( #In_Functional_Test_Even.Star_Test_PLC_Functional_Test_16 )
      Contact( #In_Functional_Test_Even.Visual_Test_Approved_PLC_Functional_Test_16 )
      S_Move(in := 'APROVADO', out => #Functional_Tests_Panels[16].Visual_Test)
   END_RUNG
   RUNG wire#powerrail
      Contact( #In_Functional_Test_Even.Star_Test_PLC_Functional_Test_16 )
      I_Contact( #In_Functional_Test_Even.Visual_Test_Approved_PLC_Functional_Test_16 )
      S_Move(in := 'REPROVADO', out => #Functional_Tests_Panels[16].Visual_Test)
   END_RUNG
   RUNG wire#powerrail
      Contact( #In_Functional_Test_Even.Star_Test_PLC_Functional_Test_16 )
      Contact( #In_Functional_Test_Even.Electrical_Current_Test_Approved_PLC_Functional_Test_16 )
      Contact( #In_Functional_Test_Even.Visual_Test_Approved_PLC_Functional_Test_16 )
      S_Move(in := 'APROVADO', out => #Functional_Tests_Panels[16].Functional_Test)
   END_RUNG
   RUNG wire#powerrail
      Contact( #In_Functional_Test_Even.Star_Test_PLC_Functional_Test_16 )
      wire#w1
      I_Contact( #In_Functional_Test_Even.Electrical_Current_Test_Approved_PLC_Functional_Test_16 )
      wire#w2
      S_Move(in := 'REPROVADO', out => #Functional_Tests_Panels[16].Functional_Test)
   END_RUNG
   RUNG wire#w1
      I_Contact( #In_Functional_Test_Even.Visual_Test_Approved_PLC_Functional_Test_16 )
   END_RUNG wire#w2
   // the same network as SCL:
   #_w1 := #In_Functional_Test_Even.Star_Test_PLC_Functional_Test_16 AND NOT #Aux_Trigger_16;   // rising edge of #In_Functional_Test_Even.Star_Test_PLC_Functional_Test_16
   #Aux_Trigger_16 := #In_Functional_Test_Even.Star_Test_PLC_Functional_Test_16;
   IF #_w1 THEN
       #Functional_Tests_Panels[16].Water_Fountain := #Water_Fountain;
       #Functional_Tests_Panels[16].Serial_Number := #Serial_Number;
   END_IF;
   IF #In_Functional_Test_Even.Star_Test_PLC_Functional_Test_16 THEN
       #Functional_Tests_Panels[16].Read_Electrical_Voltage := #Read_Electrial_Voltage;
   END_IF;
   IF #In_Functional_Test_Even.Star_Test_PLC_Functional_Test_16 AND NOT #In_Functional_Test_Even.Electrical_Current_Test_Approved_PLC_Functional_Test_16 THEN
       #Functional_Tests_Panels[16].Electrical_Current_Test := 'REPROVADO';
       #Functional_Tests_Panels[16].Read_Electrical_Current := #In_Functional_Test_Even.Electrical_Current_Read_PLC_Functional_Test_16;
   END_IF;
   IF #In_Functional_Test_Even.Star_Test_PLC_Functional_Test_16 AND #In_Functional_Test_Even.Electrical_Current_Test_Approved_PLC_Functional_Test_16 THEN
       #Functional_Tests_Panels[16].Electrical_Current_Test := 'APROVADO';
   END_IF;
   IF #In_Functional_Test_Even.Star_Test_PLC_Functional_Test_16 AND #In_Functional_Test_Even.Visual_Test_Approved_PLC_Functional_Test_16 THEN
       #Functional_Tests_Panels[16].Visual_Test := 'APROVADO';
   END_IF;
   IF #In_Functional_Test_Even.Star_Test_PLC_Functional_Test_16 AND NOT #In_Functional_Test_Even.Visual_Test_Approved_PLC_Functional_Test_16 THEN
       #Functional_Tests_Panels[16].Visual_Test := 'REPROVADO';
   END_IF;
   IF #In_Functional_Test_Even.Star_Test_PLC_Functional_Test_16 AND #In_Functional_Test_Even.Electrical_Current_Test_Approved_PLC_Functional_Test_16 AND #In_Functional_Test_Even.Visual_Test_Approved_PLC_Functional_Test_16 THEN
       #Functional_Tests_Panels[16].Functional_Test := 'APROVADO';
   END_IF;
   IF #In_Functional_Test_Even.Star_Test_PLC_Functional_Test_16 AND (NOT #In_Functional_Test_Even.Electrical_Current_Test_Approved_PLC_Functional_Test_16 OR NOT #In_Functional_Test_Even.Visual_Test_Approved_PLC_Functional_Test_16) THEN
       #Functional_Tests_Panels[16].Functional_Test := 'REPROVADO';
   END_IF;
END_REGION

REGION Network 17: Panel 17
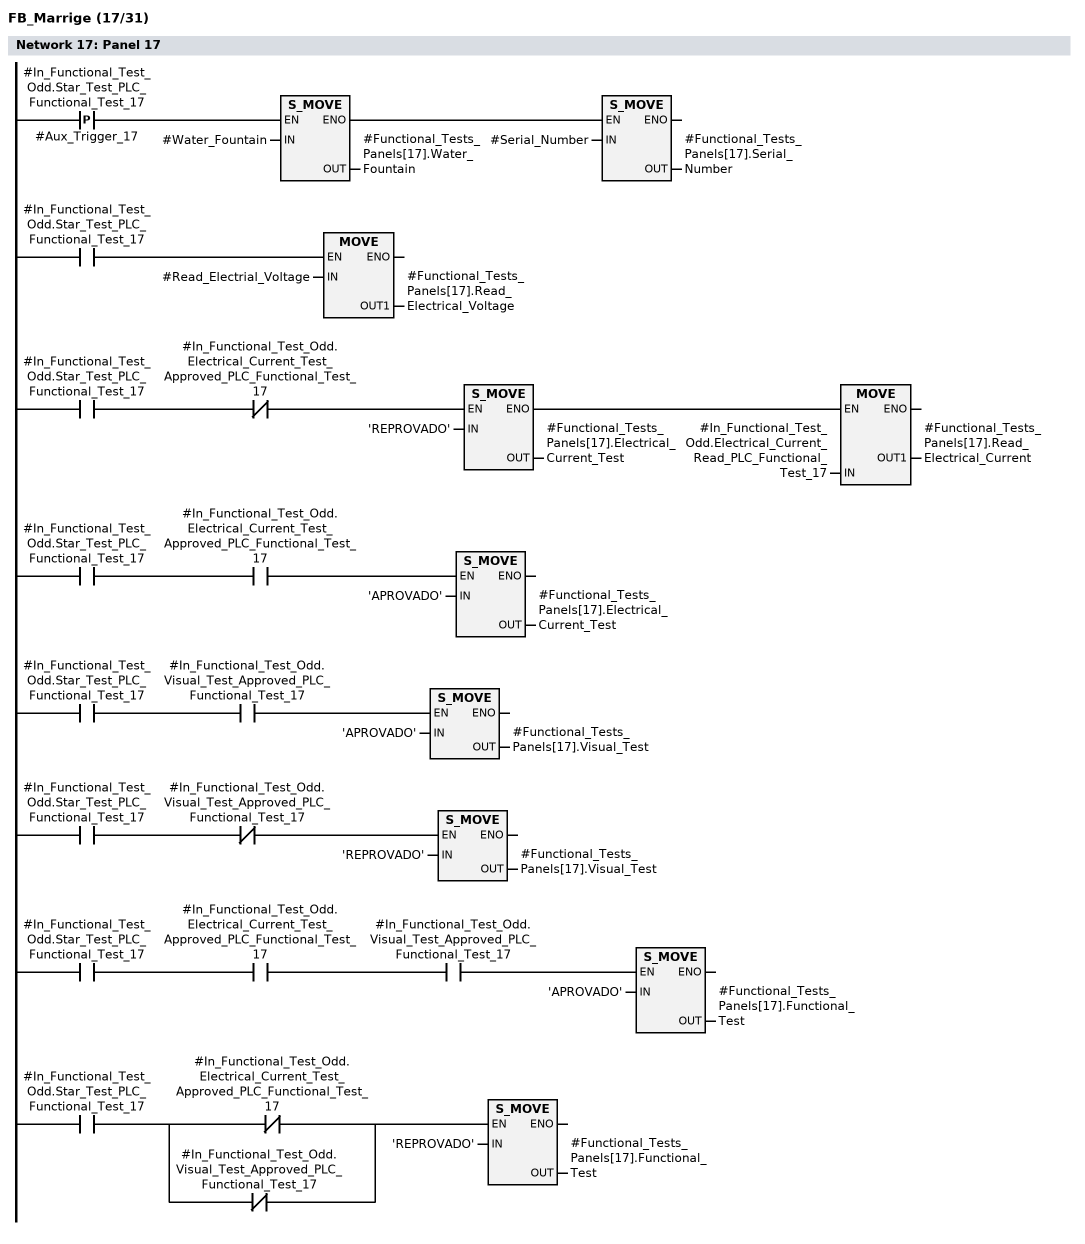
   RUNG wire#powerrail
      P_Contact(operand := #In_Functional_Test_Odd.Star_Test_PLC_Functional_Test_17, bit := #Aux_Trigger_17)
      S_Move(in := #Water_Fountain, out => #Functional_Tests_Panels[17].Water_Fountain)
      S_Move(in := #Serial_Number, out => #Functional_Tests_Panels[17].Serial_Number)
   END_RUNG
   RUNG wire#powerrail
      Contact( #In_Functional_Test_Odd.Star_Test_PLC_Functional_Test_17 )
      Move(in := #Read_Electrial_Voltage, out1 => #Functional_Tests_Panels[17].Read_Electrical_Voltage)
   END_RUNG
   RUNG wire#powerrail
      Contact( #In_Functional_Test_Odd.Star_Test_PLC_Functional_Test_17 )
      I_Contact( #In_Functional_Test_Odd.Electrical_Current_Test_Approved_PLC_Functional_Test_17 )
      S_Move(in := 'REPROVADO', out => #Functional_Tests_Panels[17].Electrical_Current_Test)
      Move(in := #In_Functional_Test_Odd.Electrical_Current_Read_PLC_Functional_Test_17, out1 => #Functional_Tests_Panels[17].Read_Electrical_Current)
   END_RUNG
   RUNG wire#powerrail
      Contact( #In_Functional_Test_Odd.Star_Test_PLC_Functional_Test_17 )
      Contact( #In_Functional_Test_Odd.Electrical_Current_Test_Approved_PLC_Functional_Test_17 )
      S_Move(in := 'APROVADO', out => #Functional_Tests_Panels[17].Electrical_Current_Test)
   END_RUNG
   RUNG wire#powerrail
      Contact( #In_Functional_Test_Odd.Star_Test_PLC_Functional_Test_17 )
      Contact( #In_Functional_Test_Odd.Visual_Test_Approved_PLC_Functional_Test_17 )
      S_Move(in := 'APROVADO', out => #Functional_Tests_Panels[17].Visual_Test)
   END_RUNG
   RUNG wire#powerrail
      Contact( #In_Functional_Test_Odd.Star_Test_PLC_Functional_Test_17 )
      I_Contact( #In_Functional_Test_Odd.Visual_Test_Approved_PLC_Functional_Test_17 )
      S_Move(in := 'REPROVADO', out => #Functional_Tests_Panels[17].Visual_Test)
   END_RUNG
   RUNG wire#powerrail
      Contact( #In_Functional_Test_Odd.Star_Test_PLC_Functional_Test_17 )
      Contact( #In_Functional_Test_Odd.Electrical_Current_Test_Approved_PLC_Functional_Test_17 )
      Contact( #In_Functional_Test_Odd.Visual_Test_Approved_PLC_Functional_Test_17 )
      S_Move(in := 'APROVADO', out => #Functional_Tests_Panels[17].Functional_Test)
   END_RUNG
   RUNG wire#powerrail
      Contact( #In_Functional_Test_Odd.Star_Test_PLC_Functional_Test_17 )
      wire#w1
      I_Contact( #In_Functional_Test_Odd.Electrical_Current_Test_Approved_PLC_Functional_Test_17 )
      wire#w2
      S_Move(in := 'REPROVADO', out => #Functional_Tests_Panels[17].Functional_Test)
   END_RUNG
   RUNG wire#w1
      I_Contact( #In_Functional_Test_Odd.Visual_Test_Approved_PLC_Functional_Test_17 )
   END_RUNG wire#w2
   // the same network as SCL:
   #_w1 := #In_Functional_Test_Odd.Star_Test_PLC_Functional_Test_17 AND NOT #Aux_Trigger_17;   // rising edge of #In_Functional_Test_Odd.Star_Test_PLC_Functional_Test_17
   #Aux_Trigger_17 := #In_Functional_Test_Odd.Star_Test_PLC_Functional_Test_17;
   IF #_w1 THEN
       #Functional_Tests_Panels[17].Water_Fountain := #Water_Fountain;
       #Functional_Tests_Panels[17].Serial_Number := #Serial_Number;
   END_IF;
   IF #In_Functional_Test_Odd.Star_Test_PLC_Functional_Test_17 THEN
       #Functional_Tests_Panels[17].Read_Electrical_Voltage := #Read_Electrial_Voltage;
   END_IF;
   IF #In_Functional_Test_Odd.Star_Test_PLC_Functional_Test_17 AND NOT #In_Functional_Test_Odd.Electrical_Current_Test_Approved_PLC_Functional_Test_17 THEN
       #Functional_Tests_Panels[17].Electrical_Current_Test := 'REPROVADO';
       #Functional_Tests_Panels[17].Read_Electrical_Current := #In_Functional_Test_Odd.Electrical_Current_Read_PLC_Functional_Test_17;
   END_IF;
   IF #In_Functional_Test_Odd.Star_Test_PLC_Functional_Test_17 AND #In_Functional_Test_Odd.Electrical_Current_Test_Approved_PLC_Functional_Test_17 THEN
       #Functional_Tests_Panels[17].Electrical_Current_Test := 'APROVADO';
   END_IF;
   IF #In_Functional_Test_Odd.Star_Test_PLC_Functional_Test_17 AND #In_Functional_Test_Odd.Visual_Test_Approved_PLC_Functional_Test_17 THEN
       #Functional_Tests_Panels[17].Visual_Test := 'APROVADO';
   END_IF;
   IF #In_Functional_Test_Odd.Star_Test_PLC_Functional_Test_17 AND NOT #In_Functional_Test_Odd.Visual_Test_Approved_PLC_Functional_Test_17 THEN
       #Functional_Tests_Panels[17].Visual_Test := 'REPROVADO';
   END_IF;
   IF #In_Functional_Test_Odd.Star_Test_PLC_Functional_Test_17 AND #In_Functional_Test_Odd.Electrical_Current_Test_Approved_PLC_Functional_Test_17 AND #In_Functional_Test_Odd.Visual_Test_Approved_PLC_Functional_Test_17 THEN
       #Functional_Tests_Panels[17].Functional_Test := 'APROVADO';
   END_IF;
   IF #In_Functional_Test_Odd.Star_Test_PLC_Functional_Test_17 AND (NOT #In_Functional_Test_Odd.Electrical_Current_Test_Approved_PLC_Functional_Test_17 OR NOT #In_Functional_Test_Odd.Visual_Test_Approved_PLC_Functional_Test_17) THEN
       #Functional_Tests_Panels[17].Functional_Test := 'REPROVADO';
   END_IF;
END_REGION

REGION Network 18: Panel 18
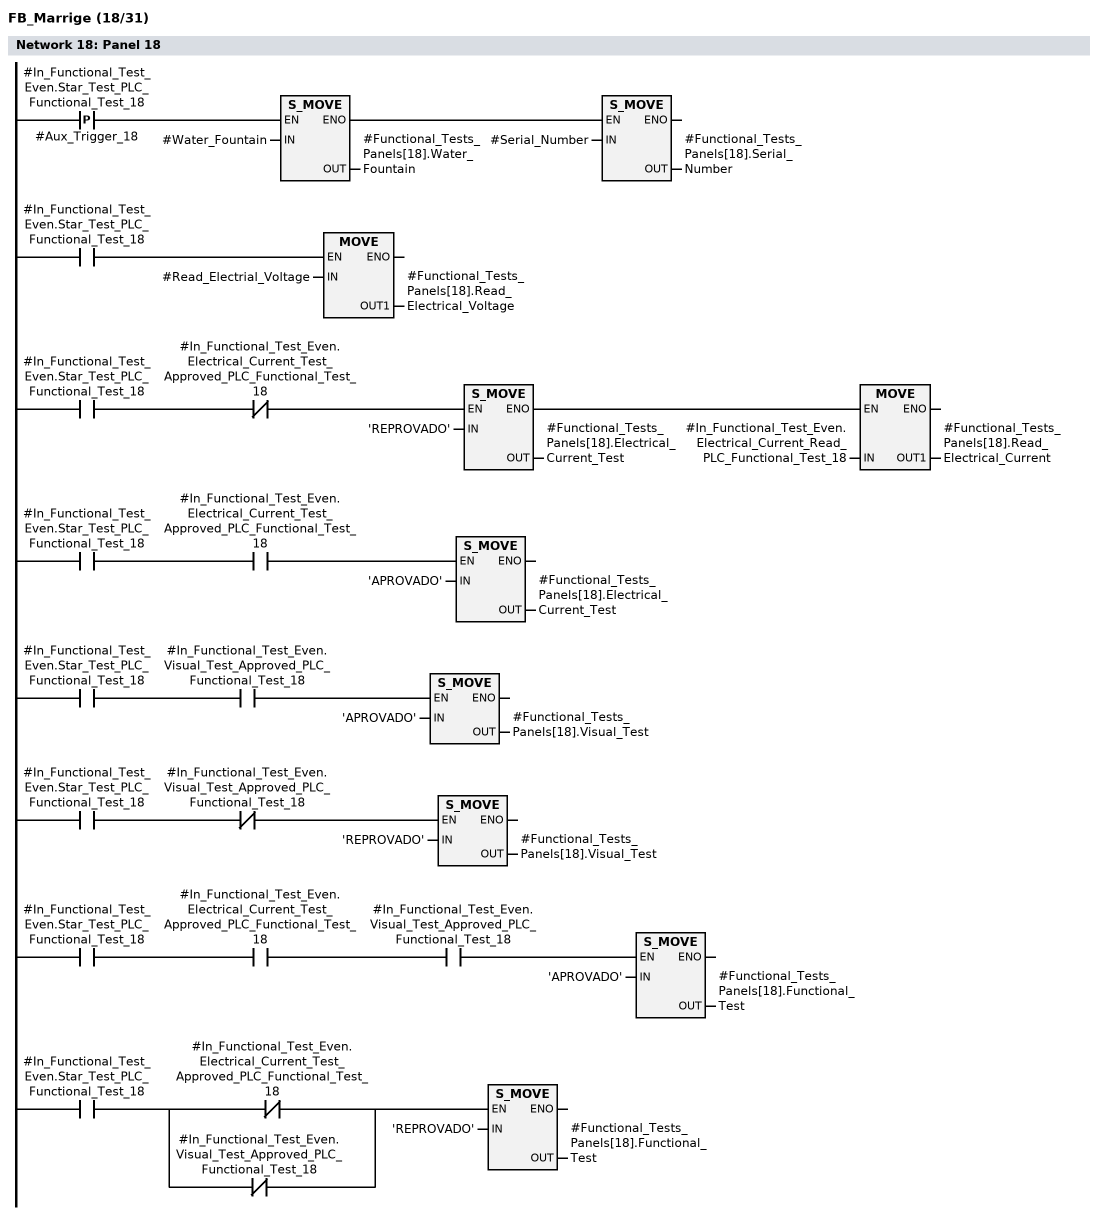
   RUNG wire#powerrail
      P_Contact(operand := #In_Functional_Test_Even.Star_Test_PLC_Functional_Test_18, bit := #Aux_Trigger_18)
      S_Move(in := #Water_Fountain, out => #Functional_Tests_Panels[18].Water_Fountain)
      S_Move(in := #Serial_Number, out => #Functional_Tests_Panels[18].Serial_Number)
   END_RUNG
   RUNG wire#powerrail
      Contact( #In_Functional_Test_Even.Star_Test_PLC_Functional_Test_18 )
      Move(in := #Read_Electrial_Voltage, out1 => #Functional_Tests_Panels[18].Read_Electrical_Voltage)
   END_RUNG
   RUNG wire#powerrail
      Contact( #In_Functional_Test_Even.Star_Test_PLC_Functional_Test_18 )
      I_Contact( #In_Functional_Test_Even.Electrical_Current_Test_Approved_PLC_Functional_Test_18 )
      S_Move(in := 'REPROVADO', out => #Functional_Tests_Panels[18].Electrical_Current_Test)
      Move(in := #In_Functional_Test_Even.Electrical_Current_Read_PLC_Functional_Test_18, out1 => #Functional_Tests_Panels[18].Read_Electrical_Current)
   END_RUNG
   RUNG wire#powerrail
      Contact( #In_Functional_Test_Even.Star_Test_PLC_Functional_Test_18 )
      Contact( #In_Functional_Test_Even.Electrical_Current_Test_Approved_PLC_Functional_Test_18 )
      S_Move(in := 'APROVADO', out => #Functional_Tests_Panels[18].Electrical_Current_Test)
   END_RUNG
   RUNG wire#powerrail
      Contact( #In_Functional_Test_Even.Star_Test_PLC_Functional_Test_18 )
      Contact( #In_Functional_Test_Even.Visual_Test_Approved_PLC_Functional_Test_18 )
      S_Move(in := 'APROVADO', out => #Functional_Tests_Panels[18].Visual_Test)
   END_RUNG
   RUNG wire#powerrail
      Contact( #In_Functional_Test_Even.Star_Test_PLC_Functional_Test_18 )
      I_Contact( #In_Functional_Test_Even.Visual_Test_Approved_PLC_Functional_Test_18 )
      S_Move(in := 'REPROVADO', out => #Functional_Tests_Panels[18].Visual_Test)
   END_RUNG
   RUNG wire#powerrail
      Contact( #In_Functional_Test_Even.Star_Test_PLC_Functional_Test_18 )
      Contact( #In_Functional_Test_Even.Electrical_Current_Test_Approved_PLC_Functional_Test_18 )
      Contact( #In_Functional_Test_Even.Visual_Test_Approved_PLC_Functional_Test_18 )
      S_Move(in := 'APROVADO', out => #Functional_Tests_Panels[18].Functional_Test)
   END_RUNG
   RUNG wire#powerrail
      Contact( #In_Functional_Test_Even.Star_Test_PLC_Functional_Test_18 )
      wire#w1
      I_Contact( #In_Functional_Test_Even.Electrical_Current_Test_Approved_PLC_Functional_Test_18 )
      wire#w2
      S_Move(in := 'REPROVADO', out => #Functional_Tests_Panels[18].Functional_Test)
   END_RUNG
   RUNG wire#w1
      I_Contact( #In_Functional_Test_Even.Visual_Test_Approved_PLC_Functional_Test_18 )
   END_RUNG wire#w2
   // the same network as SCL:
   #_w1 := #In_Functional_Test_Even.Star_Test_PLC_Functional_Test_18 AND NOT #Aux_Trigger_18;   // rising edge of #In_Functional_Test_Even.Star_Test_PLC_Functional_Test_18
   #Aux_Trigger_18 := #In_Functional_Test_Even.Star_Test_PLC_Functional_Test_18;
   IF #_w1 THEN
       #Functional_Tests_Panels[18].Water_Fountain := #Water_Fountain;
       #Functional_Tests_Panels[18].Serial_Number := #Serial_Number;
   END_IF;
   IF #In_Functional_Test_Even.Star_Test_PLC_Functional_Test_18 THEN
       #Functional_Tests_Panels[18].Read_Electrical_Voltage := #Read_Electrial_Voltage;
   END_IF;
   IF #In_Functional_Test_Even.Star_Test_PLC_Functional_Test_18 AND NOT #In_Functional_Test_Even.Electrical_Current_Test_Approved_PLC_Functional_Test_18 THEN
       #Functional_Tests_Panels[18].Electrical_Current_Test := 'REPROVADO';
       #Functional_Tests_Panels[18].Read_Electrical_Current := #In_Functional_Test_Even.Electrical_Current_Read_PLC_Functional_Test_18;
   END_IF;
   IF #In_Functional_Test_Even.Star_Test_PLC_Functional_Test_18 AND #In_Functional_Test_Even.Electrical_Current_Test_Approved_PLC_Functional_Test_18 THEN
       #Functional_Tests_Panels[18].Electrical_Current_Test := 'APROVADO';
   END_IF;
   IF #In_Functional_Test_Even.Star_Test_PLC_Functional_Test_18 AND #In_Functional_Test_Even.Visual_Test_Approved_PLC_Functional_Test_18 THEN
       #Functional_Tests_Panels[18].Visual_Test := 'APROVADO';
   END_IF;
   IF #In_Functional_Test_Even.Star_Test_PLC_Functional_Test_18 AND NOT #In_Functional_Test_Even.Visual_Test_Approved_PLC_Functional_Test_18 THEN
       #Functional_Tests_Panels[18].Visual_Test := 'REPROVADO';
   END_IF;
   IF #In_Functional_Test_Even.Star_Test_PLC_Functional_Test_18 AND #In_Functional_Test_Even.Electrical_Current_Test_Approved_PLC_Functional_Test_18 AND #In_Functional_Test_Even.Visual_Test_Approved_PLC_Functional_Test_18 THEN
       #Functional_Tests_Panels[18].Functional_Test := 'APROVADO';
   END_IF;
   IF #In_Functional_Test_Even.Star_Test_PLC_Functional_Test_18 AND (NOT #In_Functional_Test_Even.Electrical_Current_Test_Approved_PLC_Functional_Test_18 OR NOT #In_Functional_Test_Even.Visual_Test_Approved_PLC_Functional_Test_18) THEN
       #Functional_Tests_Panels[18].Functional_Test := 'REPROVADO';
   END_IF;
END_REGION

